C03680=1105.815,151.966,-63.092,-179.395,8.807,149.540
C03681=1105.819,151.717,-63.070,-179.397,8.804,149.540
C03682=1105.824,151.467,-63.048,-179.399,8.800,149.540
C03683=1105.829,151.219,-63.025,-179.401,8.797,149.539
C03684=1105.833,150.970,-63.003,-179.403,8.794,149.539
C03685=1105.838,150.721,-62.980,-179.405,8.790,149.539
C03686=1105.843,150.472,-62.958,-179.407,8.787,149.539
C03687=1105.847,150.223,-62.936,-179.409,8.783,149.538
C03688=1105.852,149.974,-62.913,-179.410,8.781,149.538
C03689=1105.856,149.725,-62.891,-179.413,8.777,149.538
C03690=1105.861,149.476,-62.869,-179.415,8.774,149.538
C03691=1105.865,149.228,-62.847,-179.417,8.770,149.537
C03692=1105.870,148.978,-62.824,-179.418,8.766,149.537
C03693=1105.875,148.729,-62.802,-179.420,8.764,149.537
C03694=1105.879,148.480,-62.780,-179.422,8.760,149.536
C03695=1105.883,148.231,-62.757,-179.424,8.757,149.536
C03696=1105.889,147.982,-62.735,-179.426,8.753,149.536
C03697=1105.893,147.733,-62.713,-179.428,8.749,149.536
C03698=1105.898,147.484,-62.691,-179.430,8.746,149.535
C03699=1105.902,147.236,-62.669,-179.431,8.743,149.535
C03700=1105.908,146.987,-62.646,-179.433,8.740,149.535
C03701=1105.911,146.773,-62.628,-179.435,8.736,149.535
C03702=1105.915,146.560,-62.608,-179.436,8.733,149.534
C03703=1105.919,146.347,-62.590,-179.438,8.730,149.534
C03704=1105.923,146.133,-62.570,-179.439,8.728,149.534
C03705=1105.927,145.920,-62.552,-179.441,8.724,149.533
C03706=1105.931,145.707,-62.533,-179.443,8.721,149.533
C03707=1105.935,145.493,-62.514,-179.444,8.719,149.533
C03708=1105.939,145.280,-62.495,-179.446,8.715,149.533
C03709=1105.943,145.031,-62.473,-179.448,8.711,149.532
C03710=1105.948,144.782,-62.451,-179.449,8.708,149.532
C03711=1105.953,144.533,-62.429,-179.451,8.705,149.532
C03712=1105.957,144.284,-62.408,-179.453,8.701,149.531
C03713=1105.962,144.035,-62.385,-179.455,8.697,149.531
C03714=1105.967,143.787,-62.364,-179.456,8.695,149.531
C03715=1105.972,143.537,-62.341,-179.458,8.691,149.530
C03716=1105.976,143.288,-62.319,-179.460,8.687,149.530
C03717=1105.981,143.039,-62.297,-179.462,8.683,149.530
C03718=1105.986,142.790,-62.276,-179.464,8.680,149.529
C03719=1105.990,142.541,-62.254,-179.465,8.677,149.529
C03720=1105.995,142.292,-62.232,-179.467,8.673,149.529
C03721=1105.999,142.043,-62.210,-179.469,8.670,149.528
C03722=1106.004,141.794,-62.188,-179.470,8.666,149.528
C03723=1106.009,141.546,-62.167,-179.472,8.663,149.528
C03724=1106.013,141.296,-62.145,-179.474,8.660,149.528
C03725=1106.018,141.048,-62.123,-179.476,8.656,149.527
C03726=1106.022,140.798,-62.101,-179.478,8.652,149.527
C03727=1106.027,140.550,-62.079,-179.479,8.650,149.527
C03728=1106.031,140.300,-62.057,-179.481,8.646,149.526
C03729=1106.036,140.052,-62.035,-179.483,8.642,149.526
C03730=1106.040,139.802,-62.013,-179.485,8.639,149.526
C03731=1106.046,139.553,-61.992,-179.486,8.636,149.525
C03732=1106.050,139.304,-61.971,-179.488,8.632,149.525
C03733=1106.055,139.055,-61.949,-179.490,8.629,149.525
C03734=1106.060,138.806,-61.927,-179.491,8.626,149.524
C03735=1106.064,138.557,-61.905,-179.493,8.622,149.524
C03736=1106.069,138.308,-61.883,-179.495,8.619,149.524
C03737=1106.074,138.059,-61.862,-179.497,8.615,149.523
C03738=1106.078,137.810,-61.840,-179.498,8.612,149.523
C03739=1106.082,137.562,-61.819,-179.500,8.609,149.523
C03740=1106.087,137.312,-61.797,-179.502,8.605,149.523
C03741=1106.092,137.063,-61.776,-179.504,8.601,149.522
C03742=1106.097,136.814,-61.754,-179.505,8.599,149.522
C03743=1106.101,136.565,-61.732,-179.507,8.595,149.522
C03744=1106.106,136.316,-61.711,-179.509,8.591,149.521
C03745=1106.111,136.067,-61.690,-179.511,8.589,149.521
C03746=1106.115,135.818,-61.668,-179.512,8.585,149.521
C03747=1106.120,135.569,-61.646,-179.514,8.581,149.521
C03748=1106.125,135.320,-61.626,-179.516,8.578,149.520
C03749=1106.129,135.071,-61.604,-179.518,8.575,149.520
C03750=1106.134,134.822,-61.582,-179.519,8.571,149.520
C03751=1106.139,134.573,-61.561,-179.522,8.568,149.519
C03752=1106.143,134.324,-61.539,-179.523,8.565,149.519
C03753=1106.148,134.075,-61.517,-179.525,8.561,149.519
C03754=1106.152,133.826,-61.497,-179.527,8.558,149.518
C03755=1106.157,133.577,-61.475,-179.529,8.554,149.518
C03756=1106.162,133.327,-61.454,-179.530,8.551,149.518
C03757=1106.166,133.114,-61.436,-179.532,8.549,149.518
C03758=1106.170,132.901,-61.418,-179.533,8.545,149.517
C03759=1106.174,132.688,-61.399,-179.535,8.542,149.517
C03760=1106.178,132.474,-61.381,-179.536,8.539,149.517
C03761=1106.182,132.261,-61.362,-179.538,8.537,149.517
C03762=1106.186,132.047,-61.344,-179.539,8.534,149.516
C03763=1106.190,131.834,-61.326,-179.540,8.531,149.516
C03764=1106.194,131.621,-61.308,-179.543,8.528,149.516
C03765=1106.199,131.372,-61.287,-179.544,8.525,149.516
C03766=1106.203,131.122,-61.265,-179.546,8.521,149.516
C03767=1106.208,130.873,-61.244,-179.548,8.518,149.515
C03768=1106.212,130.625,-61.223,-179.549,8.515,149.515
C03769=1106.217,130.376,-61.202,-179.551,8.511,149.515
C03770=1106.222,130.126,-61.180,-179.553,8.508,149.514
C03771=1106.226,129.877,-61.159,-179.554,8.505,149.514
C03772=1106.231,129.629,-61.138,-179.556,8.501,149.514
C03773=1106.236,129.379,-61.117,-179.558,8.498,149.513
C03774=1106.241,129.130,-61.096,-179.560,8.495,149.513
C03775=1106.245,128.881,-61.074,-179.561,8.491,149.513
C03776=1106.250,128.632,-61.053,-179.564,8.488,149.513
C03777=1106.255,128.383,-61.033,-179.566,8.484,149.512
C03778=1106.259,128.134,-61.011,-179.567,8.481,149.512
C03779=1106.265,127.885,-60.990,-179.569,8.478,149.512
C03780=1106.268,127.635,-60.970,-179.571,8.474,149.511
C03781=1106.273,127.387,-60.948,-179.572,8.471,149.511
C03782=1106.278,127.137,-60.927,-179.574,8.468,149.511
C03783=1106.283,126.889,-60.907,-179.576,8.464,149.511
C03784=1106.288,126.640,-60.885,-179.577,8.461,149.510
C03785=1106.292,126.391,-60.865,-179.579,8.458,149.510
C03786=1106.297,126.141,-60.843,-179.581,8.454,149.510
C03787=1106.302,125.892,-60.822,-179.582,8.451,149.509
C03788=1106.306,125.643,-60.801,-179.585,8.448,149.509
C03789=1106.311,125.394,-60.780,-179.587,8.444,149.509
C03790=1106.316,125.145,-60.760,-179.588,8.442,149.509
C03791=1106.321,124.896,-60.739,-179.590,8.438,149.508
C03792=1106.325,124.648,-60.718,-179.592,8.434,149.508
C03793=1106.330,124.398,-60.696,-179.593,8.431,149.508
C03794=1106.334,124.149,-60.676,-179.595,8.428,149.508
C03795=1106.339,123.899,-60.655,-179.597,8.424,149.507
C03796=1106.344,123.650,-60.635,-179.598,8.421,149.507
C03797=1106.349,123.401,-60.614,-179.600,8.418,149.507
C03798=1106.353,123.153,-60.593,-179.602,8.414,149.506
C03799=1106.358,122.904,-60.572,-179.603,8.411,149.506
C03800=1106.363,122.655,-60.551,-179.605,8.408,149.506
C03801=1106.368,122.405,-60.530,-179.608,8.404,149.506
C03802=1106.372,122.156,-60.510,-179.609,8.402,149.505
C03803=1106.376,121.907,-60.489,-179.611,8.398,149.505
C03804=1106.381,121.658,-60.468,-179.613,8.394,149.505
C03805=1106.386,121.409,-60.448,-179.614,8.391,149.504
C03806=1106.391,121.159,-60.427,-179.616,8.388,149.504
C03807=1106.395,120.910,-60.407,-179.618,8.384,149.504
C03808=1106.400,120.661,-60.386,-179.620,8.381,149.504
C03809=1106.405,120.412,-60.365,-179.621,8.378,149.503
C03810=1106.409,120.163,-60.345,-179.623,8.374,149.503
C03811=1106.414,119.914,-60.324,-179.625,8.370,149.503
C03812=1106.419,119.665,-60.304,-179.626,8.368,149.502
C03813=1106.423,119.452,-60.285,-179.628,8.365,149.502
C03814=1106.427,119.238,-60.268,-179.630,8.362,149.502
C03815=1106.431,119.025,-60.250,-179.631,8.359,149.502
C03816=1106.435,118.811,-60.232,-179.633,8.356,149.502
C03817=1106.439,118.598,-60.216,-179.634,8.353,149.501
C03818=1106.443,118.385,-60.198,-179.635,8.350,149.501
C03819=1106.447,118.171,-60.180,-179.637,8.348,149.501
C03820=1106.451,117.958,-60.162,-179.638,8.345,149.500
C03821=1106.456,117.708,-60.142,-179.640,8.341,149.500
C03822=1106.461,117.459,-60.121,-179.642,8.338,149.500
C03823=1106.465,117.210,-60.101,-179.644,8.334,149.500
C03824=1106.470,116.961,-60.081,-179.645,8.331,149.499
C03825=1106.475,116.712,-60.060,-179.647,8.328,149.499
C03826=1106.479,116.463,-60.039,-179.649,8.324,149.499
C03827=1106.484,116.214,-60.019,-179.650,8.321,149.498
C03828=1106.488,115.964,-59.999,-179.652,8.318,149.498
C03829=1106.494,115.715,-59.978,-179.654,8.314,149.498
C03830=1106.498,115.466,-59.958,-179.655,8.311,149.498
C03831=1106.503,115.218,-59.938,-179.658,8.308,149.497
C03832=1106.508,114.969,-59.918,-179.659,8.304,149.497
C03833=1106.513,114.719,-59.897,-179.661,8.301,149.497
C03834=1106.518,114.470,-59.877,-179.663,8.297,149.496
C03835=1106.522,114.221,-59.857,-179.664,8.294,149.496
C03836=1106.526,113.972,-59.836,-179.666,8.291,149.496
C03837=1106.532,113.722,-59.816,-179.668,8.287,149.496
C03838=1106.536,113.473,-59.796,-179.669,8.283,149.495
C03839=1106.541,113.224,-59.775,-179.671,8.280,149.495
C03840=1106.545,112.975,-59.756,-179.672,8.277,149.494
C03841=1106.550,112.726,-59.735,-179.674,8.273,149.494
C03842=1106.555,112.476,-59.714,-179.677,8.270,149.494
C03843=1106.560,112.228,-59.695,-179.678,8.267,149.494
C03844=1106.565,111.979,-59.675,-179.680,8.263,149.493
C03845=1106.569,111.730,-59.654,-179.681,8.259,149.493
C03846=1106.574,111.480,-59.634,-179.683,8.257,149.493
C03847=1106.578,111.231,-59.614,-179.685,8.253,149.492
C03848=1106.583,110.982,-59.594,-179.686,8.249,149.492
C03849=1106.588,110.732,-59.573,-179.688,8.246,149.492
C03850=1106.593,110.484,-59.553,-179.690,8.242,149.492
C03851=1106.598,110.235,-59.534,-179.692,8.238,149.491
C03852=1106.603,109.986,-59.513,-179.694,8.235,149.491
C03853=1106.607,109.736,-59.494,-179.696,8.231,149.491
C03854=1106.612,109.487,-59.473,-179.698,8.228,149.490
C03855=1106.617,109.237,-59.454,-179.699,8.225,149.490
C03856=1106.622,108.989,-59.434,-179.701,8.221,149.490
C03857=1106.626,108.740,-59.414,-179.703,8.217,149.489
C03858=1106.631,108.491,-59.394,-179.705,8.214,149.489
C03859=1106.636,108.241,-59.374,-179.706,8.210,149.489
C03860=1106.640,107.992,-59.354,-179.709,8.207,149.488
C03861=1106.645,107.743,-59.334,-179.710,8.203,149.488
C03862=1106.650,107.494,-59.315,-179.712,8.199,149.488
C03863=1106.654,107.245,-59.294,-179.714,8.195,149.487
C03864=1106.659,106.995,-59.275,-179.716,8.192,149.487
C03865=1106.664,106.746,-59.254,-179.717,8.188,149.487
C03866=1106.669,106.497,-59.235,-179.719,8.185,149.486
C03867=1106.674,106.248,-59.215,-179.721,8.181,149.486
C03868=1106.678,105.999,-59.195,-179.723,8.178,149.486
C03869=1106.682,105.785,-59.178,-179.724,8.174,149.485
C03870=1106.686,105.572,-59.161,-179.726,8.171,149.485
C03871=1106.691,105.358,-59.144,-179.727,8.168,149.485
C03872=1106.695,105.144,-59.127,-179.729,8.165,149.484
C03873=1106.699,104.931,-59.110,-179.730,8.162,149.484
C03874=1106.703,104.717,-59.093,-179.731,8.159,149.484
C03875=1106.707,104.504,-59.076,-179.733,8.155,149.484
C03876=1106.711,104.290,-59.059,-179.734,8.152,149.483
C03877=1106.715,104.041,-59.040,-179.736,8.149,149.483
C03878=1106.720,103.792,-59.020,-179.738,8.145,149.482
C03879=1106.726,103.543,-59.001,-179.739,8.142,149.482
C03880=1106.730,103.294,-58.981,-179.741,8.138,149.482
C03881=1106.735,103.044,-58.961,-179.742,8.134,149.481
C03882=1106.740,102.795,-58.942,-179.744,8.130,149.481
C03883=1106.745,102.546,-58.922,-179.746,8.126,149.480
C03884=1106.749,102.297,-58.902,-179.747,8.123,149.480
C03885=1106.753,102.048,-58.883,-179.749,8.119,149.480
C03886=1106.759,101.799,-58.863,-179.751,8.115,149.479
C03887=1106.763,101.549,-58.844,-179.752,8.112,149.479
C03888=1106.768,101.299,-58.824,-179.753,8.108,149.479
C03889=1106.773,101.051,-58.805,-179.755,8.104,149.478
C03890=1106.778,100.802,-58.784,-179.757,8.100,149.478
C03891=1106.782,100.552,-58.765,-179.759,8.097,149.477
C03892=1106.787,100.304,-58.746,-179.760,8.093,149.477
C03893=1106.792,100.054,-58.726,-179.761,8.090,149.477
C03894=1106.797,99.805,-58.707,-179.763,8.086,149.476
C03895=1106.802,99.556,-58.687,-179.764,8.082,149.476
C03896=1106.806,99.306,-58.668,-179.766,8.078,149.475
C03897=1106.811,99.057,-58.649,-179.768,8.074,149.475
C03898=1106.816,98.808,-58.629,-179.769,8.070,149.474
C03899=1106.821,98.558,-58.610,-179.770,8.067,149.474
C03900=1106.825,98.310,-58.591,-179.772,8.063,149.473
C03901=1106.830,98.060,-58.571,-179.773,8.060,149.473
C03902=1106.836,97.811,-58.552,-179.775,8.056,149.473
C03903=1106.840,97.562,-58.533,-179.777,8.052,149.472
C03904=1106.844,97.312,-58.513,-179.778,8.049,149.472
C03905=1106.850,97.064,-58.494,-179.779,8.045,149.471
C03906=1106.854,96.814,-58.474,-179.781,8.041,149.471
C03907=1106.859,96.565,-58.456,-179.782,8.037,149.470
C03908=1106.864,96.316,-58.436,-179.784,8.033,149.470
C03909=1106.869,96.066,-58.416,-179.785,8.030,149.470
C03910=1106.873,95.818,-58.398,-179.787,8.026,149.469
C03911=1106.878,95.568,-58.378,-179.788,8.022,149.469
C03912=1106.883,95.319,-58.359,-179.790,8.018,149.468
C03913=1106.887,95.070,-58.340,-179.791,8.014,149.468
C03914=1106.893,94.821,-58.321,-179.792,8.011,149.467
C03915=1106.897,94.571,-58.302,-179.794,8.007,149.467
C03916=1106.902,94.322,-58.283,-179.795,8.003,149.466
C03917=1106.907,94.073,-58.263,-179.797,7.999,149.466
C03918=1106.912,93.824,-58.244,-179.798,7.996,149.465
C03919=1106.916,93.575,-58.225,-179.799,7.992,149.465
C03920=1106.921,93.325,-58.206,-179.800,7.988,149.464
C03921=1106.926,93.076,-58.187,-179.802,7.984,149.464
C03922=1106.931,92.826,-58.167,-179.803,7.981,149.463
C03923=1106.935,92.578,-58.149,-179.805,7.977,149.463
C03924=1106.940,92.328,-58.129,-179.806,7.973,149.462
C03925=1106.944,92.115,-58.113,-179.807,7.970,149.462
C03926=1106.948,91.901,-58.097,-179.808,7.967,149.462
C03927=1106.952,91.688,-58.081,-179.809,7.964,149.461
C03928=1106.957,91.474,-58.064,-179.811,7.960,149.461
C03929=1106.961,91.260,-58.048,-179.812,7.957,149.460
C03930=1106.965,91.047,-58.032,-179.813,7.954,149.460
C03931=1106.969,90.833,-58.015,-179.814,7.951,149.460
C03932=1106.973,90.619,-58.000,-179.815,7.948,149.459
C03933=1106.978,90.370,-57.980,-179.816,7.944,149.459
C03934=1106.983,90.121,-57.962,-179.817,7.940,149.458
C03935=1106.988,89.871,-57.942,-179.819,7.936,149.458
C03936=1106.992,89.622,-57.924,-179.820,7.933,149.457
C03937=1106.998,89.373,-57.905,-179.821,7.928,149.457
C03938=1107.002,89.124,-57.886,-179.823,7.924,149.456
C03939=1107.007,88.875,-57.867,-179.824,7.921,149.456
C03940=1107.011,88.625,-57.848,-179.825,7.917,149.455
C03941=1107.017,88.376,-57.829,-179.826,7.913,149.455
C03942=1107.021,88.127,-57.810,-179.827,7.910,149.454
C03943=1107.026,87.877,-57.792,-179.828,7.906,149.453
C03944=1107.031,87.629,-57.773,-179.830,7.902,149.453
C03945=1107.035,87.379,-57.755,-179.831,7.899,149.453
C03946=1107.041,87.130,-57.735,-179.832,7.894,149.452
C03947=1107.045,86.880,-57.717,-179.834,7.891,149.452
C03948=1107.050,86.631,-57.698,-179.834,7.887,149.451
C03949=1107.055,86.382,-57.680,-179.836,7.883,149.450
C03950=1107.059,86.133,-57.661,-179.837,7.879,149.450
C03951=1107.065,85.883,-57.642,-179.838,7.876,149.449
C03952=1107.069,85.634,-57.623,-179.840,7.872,149.449
C03953=1107.075,85.385,-57.604,-179.840,7.868,149.448
C03954=1107.079,85.136,-57.586,-179.842,7.864,149.448
C03955=1107.083,84.886,-57.567,-179.843,7.860,149.447
C03956=1107.089,84.637,-57.548,-179.844,7.857,149.447
C03957=1107.094,84.388,-57.530,-179.845,7.853,149.446
C03958=1107.098,84.139,-57.511,-179.846,7.850,149.446
C03959=1107.103,83.889,-57.492,-179.847,7.846,149.445
C03960=1107.107,83.640,-57.473,-179.849,7.842,149.445
C03961=1107.112,83.391,-57.455,-179.849,7.838,149.444
C03962=1107.118,83.142,-57.437,-179.851,7.834,149.444
C03963=1107.122,82.892,-57.418,-179.852,7.831,149.443
C03964=1107.127,82.643,-57.400,-179.853,7.827,149.442
C03965=1107.132,82.394,-57.382,-179.854,7.824,149.442
C03966=1107.137,82.144,-57.362,-179.855,7.819,149.441
C03967=1107.141,81.895,-57.344,-179.856,7.815,149.441
C03968=1107.146,81.647,-57.325,-179.857,7.812,149.440
C03969=1107.152,81.397,-57.307,-179.858,7.808,149.440
C03970=1107.156,81.147,-57.288,-179.859,7.805,149.439
C03971=1107.161,80.898,-57.271,-179.861,7.801,149.439
C03972=1107.166,80.650,-57.252,-179.861,7.797,149.438
C03973=1107.171,80.399,-57.233,-179.863,7.793,149.438
C03974=1107.176,80.150,-57.215,-179.863,7.790,149.437
C03975=1107.180,79.902,-57.196,-179.864,7.786,149.436
C03976=1107.185,79.652,-57.178,-179.865,7.782,149.436
C03977=1107.189,79.403,-57.160,-179.866,7.778,149.435
C03978=1107.195,79.153,-57.141,-179.867,7.775,149.435
C03979=1107.200,78.905,-57.123,-179.868,7.771,149.434
C03980=1107.204,78.655,-57.104,-179.869,7.768,149.434
C03981=1107.208,78.441,-57.089,-179.870,7.764,149.433
C03982=1107.213,78.228,-57.073,-179.871,7.761,149.433
C03983=1107.217,78.013,-57.057,-179.872,7.758,149.432
C03984=1107.221,77.800,-57.042,-179.873,7.755,149.432
C03985=1107.225,77.586,-57.026,-179.874,7.752,149.431
C03986=1107.229,77.373,-57.010,-179.874,7.748,149.431
C03987=1107.233,77.159,-56.995,-179.875,7.745,149.430
C03988=1107.237,76.944,-56.979,-179.876,7.742,149.430
C03989=1107.242,76.696,-56.961,-179.878,7.738,149.429
C03990=1107.247,76.447,-56.943,-179.879,7.734,149.429
C03991=1107.252,76.197,-56.924,-179.880,7.730,149.428
C03992=1107.257,75.947,-56.906,-179.882,7.726,149.428
C03993=1107.262,75.698,-56.888,-179.884,7.722,149.427
C03994=1107.267,75.449,-56.870,-179.885,7.718,149.427
C03995=1107.272,75.200,-56.852,-179.886,7.715,149.426
C03996=1107.276,74.951,-56.834,-179.887,7.711,149.426
C03997=1107.281,74.701,-56.815,-179.888,7.706,149.425
C03998=1107.285,74.452,-56.797,-179.890,7.703,149.425
C03999=1107.290,74.203,-56.779,-179.892,7.699,149.424
C04000=1107.295,73.954,-56.761,-179.893,7.695,149.424
C04001=1107.300,73.705,-56.743,-179.894,7.690,149.423
C04002=1107.305,73.455,-56.724,-179.896,7.687,149.423
C04003=1107.310,73.205,-56.706,-179.897,7.683,149.422
C04004=1107.315,72.956,-56.688,-179.899,7.678,149.422
C04005=1107.320,72.707,-56.670,-179.899,7.675,149.421
C04006=1107.325,72.458,-56.652,-179.901,7.671,149.421
C04007=1107.330,72.209,-56.634,-179.902,7.667,149.420
C04008=1107.335,71.959,-56.617,-179.904,7.663,149.420
C04009=1107.339,71.709,-56.598,-179.905,7.659,149.419
C04010=1107.344,71.460,-56.580,-179.906,7.655,149.419
C04011=1107.349,71.211,-56.562,-179.908,7.651,149.418
C04012=1107.354,70.961,-56.544,-179.910,7.647,149.418
C04013=1107.359,70.712,-56.526,-179.911,7.643,149.417
C04014=1107.364,70.463,-56.508,-179.912,7.640,149.417
C04015=1107.368,70.214,-56.491,-179.913,7.636,149.416
C04016=1107.373,69.965,-56.473,-179.914,7.632,149.416
C04017=1107.378,69.716,-56.455,-179.916,7.628,149.415
C04018=1107.382,69.465,-56.438,-179.917,7.624,149.415
C04019=1107.387,69.216,-56.420,-179.919,7.620,149.414
C04020=1107.392,68.967,-56.402,-179.920,7.616,149.414
C04021=1107.397,68.718,-56.384,-179.921,7.613,149.413
C04022=1107.402,68.469,-56.366,-179.922,7.608,149.413
C04023=1107.407,68.219,-56.348,-179.924,7.604,149.412
C04024=1107.412,67.970,-56.330,-179.925,7.600,149.412
C04025=1107.417,67.721,-56.312,-179.926,7.596,149.411
C04026=1107.421,67.472,-56.295,-179.928,7.592,149.411
C04027=1107.427,67.222,-56.278,-179.930,7.588,149.410
C04028=1107.431,66.973,-56.260,-179.930,7.585,149.410
C04029=1107.436,66.724,-56.242,-179.932,7.581,149.409
C04030=1107.441,66.474,-56.224,-179.933,7.577,149.409
C04031=1107.446,66.225,-56.207,-179.934,7.573,149.408
C04032=1107.451,65.976,-56.189,-179.936,7.569,149.408
C04033=1107.456,65.727,-56.171,-179.937,7.565,149.407
C04034=1107.461,65.477,-56.154,-179.939,7.561,149.407
C04035=1107.466,65.228,-56.136,-179.939,7.557,149.406
C04036=1107.471,64.978,-56.118,-179.941,7.553,149.406
C04037=1107.474,64.764,-56.103,-179.942,7.549,149.405
C04038=1107.479,64.550,-56.088,-179.943,7.546,149.405
C04039=1107.482,64.337,-56.073,-179.944,7.543,149.404
C04040=1107.487,64.123,-56.058,-179.945,7.540,149.404
C04041=1107.492,63.909,-56.043,-179.947,7.536,149.403
C04042=1107.495,63.695,-56.027,-179.948,7.533,149.403
C04043=1107.500,63.481,-56.012,-179.948,7.529,149.402
C04044=1107.504,63.267,-55.998,-179.950,7.526,149.402
C04045=1107.509,63.018,-55.980,-179.951,7.522,149.401
C04046=1107.514,62.768,-55.963,-179.952,7.518,149.401
C04047=1107.518,62.520,-55.945,-179.953,7.514,149.400
C04048=1107.523,62.270,-55.928,-179.955,7.510,149.400
C04049=1107.528,62.021,-55.910,-179.956,7.506,149.399
C04050=1107.533,61.771,-55.893,-179.957,7.502,149.399
C04051=1107.537,61.522,-55.875,-179.958,7.499,149.398
C04052=1107.543,61.272,-55.858,-179.959,7.495,149.398
C04053=1107.548,61.023,-55.840,-179.961,7.490,149.397
C04054=1107.552,60.773,-55.824,-179.962,7.486,149.397
C04055=1107.558,60.525,-55.806,-179.963,7.482,149.396
C04056=1107.563,60.275,-55.789,-179.964,7.479,149.396
C04057=1107.567,60.026,-55.771,-179.965,7.475,149.395
C04058=1107.572,59.776,-55.754,-179.967,7.471,149.394
C04059=1107.576,59.528,-55.737,-179.968,7.467,149.394
C04060=1107.582,59.278,-55.719,-179.969,7.463,149.393
C04061=1107.587,59.028,-55.702,-179.970,7.459,149.393
C04062=1107.591,58.779,-55.685,-179.972,7.455,149.392
C04063=1107.596,58.529,-55.667,-179.973,7.451,149.392
C04064=1107.601,58.280,-55.649,-179.974,7.447,149.391
C04065=1107.606,58.031,-55.633,-179.975,7.443,149.391
C04066=1107.611,57.782,-55.616,-179.977,7.439,149.390
C04067=1107.616,57.533,-55.599,-179.977,7.435,149.389
C04068=1107.621,57.283,-55.581,-179.979,7.431,149.389
C04069=1107.626,57.033,-55.564,-179.980,7.427,149.388
C04070=1107.630,56.784,-55.547,-179.982,7.423,149.388
C04071=1107.636,56.535,-55.530,-179.983,7.419,149.387
C04072=1107.640,56.286,-55.513,-179.984,7.416,149.387
C04073=1107.646,56.036,-55.496,-179.985,7.412,149.386
C04074=1107.650,55.787,-55.478,-179.986,7.407,149.386
C04075=1107.655,55.537,-55.461,-179.987,7.403,149.385
C04076=1107.660,55.288,-55.444,-179.988,7.400,149.384
C04077=1107.665,55.039,-55.428,-179.989,7.396,149.384
C04078=1107.670,54.790,-55.410,-179.990,7.392,149.383
C04079=1107.675,54.540,-55.393,-179.992,7.388,149.383
C04080=1107.679,54.291,-55.376,-179.993,7.383,149.382
C04081=1107.684,54.041,-55.359,-179.994,7.380,149.382
C04082=1107.690,53.792,-55.343,-179.995,7.376,149.381
C04083=1107.694,53.543,-55.325,-179.996,7.372,149.381
C04084=1107.699,53.293,-55.308,-179.998,7.368,149.380
C04085=1107.704,53.044,-55.291,-179.999,7.363,149.379
C04086=1107.709,52.795,-55.274,-179.999,7.360,149.379
C04087=1107.714,52.545,-55.257,179.999,7.356,149.378
C04088=1107.719,52.295,-55.241,179.998,7.352,149.378
C04089=1107.724,52.046,-55.223,179.997,7.347,149.377
C04090=1107.728,51.797,-55.206,179.996,7.344,149.377
C04091=1107.734,51.548,-55.189,179.995,7.340,149.376
C04092=1107.739,51.298,-55.172,179.994,7.336,149.375
C04093=1107.743,51.085,-55.158,179.993,7.333,149.375
C04094=1107.747,50.870,-55.144,179.991,7.329,149.374
C04095=1107.752,50.656,-55.129,179.990,7.326,149.374
C04096=1107.756,50.442,-55.115,179.990,7.322,149.373
C04097=1107.760,50.229,-55.100,179.989,7.319,149.373
C04098=1107.764,50.015,-55.086,179.988,7.316,149.372
C04099=1107.769,49.800,-55.072,179.987,7.312,149.372
C04100=1107.773,49.587,-55.057,179.986,7.308,149.371
C04101=1107.777,49.337,-55.041,179.985,7.304,149.371
C04102=1107.782,49.087,-55.023,179.984,7.301,149.370
C04103=1107.787,48.839,-55.007,179.983,7.297,149.370
C04104=1107.792,48.589,-54.990,179.982,7.292,149.369
C04105=1107.797,48.339,-54.973,179.980,7.288,149.369
C04106=1107.802,48.091,-54.957,179.979,7.284,149.368
C04107=1107.807,47.841,-54.940,179.979,7.281,149.367
C04108=1107.811,47.592,-54.923,179.978,7.276,149.367
C04109=1107.816,47.342,-54.906,179.976,7.272,149.366
C04110=1107.821,47.093,-54.890,179.975,7.268,149.365
C04111=1107.826,46.844,-54.873,179.975,7.265,149.365
C04112=1107.831,46.594,-54.856,179.974,7.260,149.364
C04113=1107.837,46.344,-54.840,179.972,7.256,149.364
C04114=1107.841,46.095,-54.824,179.971,7.252,149.363
C04115=1107.845,45.845,-54.807,179.970,7.249,149.362
C04116=1107.851,45.596,-54.790,179.969,7.244,149.362
C04117=1107.856,45.347,-54.773,179.968,7.240,149.361
C04118=1107.861,45.098,-54.757,179.967,7.236,149.361
C04119=1107.865,44.849,-54.740,179.966,7.233,149.360
C04120=1107.871,44.598,-54.724,179.965,7.228,149.359
C04121=1107.876,44.349,-54.708,179.964,7.224,149.359
C04122=1107.880,44.100,-54.691,179.963,7.220,149.358
C04123=1107.885,43.850,-54.674,179.962,7.217,149.358
C04124=1107.890,43.602,-54.658,179.961,7.212,149.357
C04125=1107.896,43.351,-54.641,179.960,7.208,149.356
C04126=1107.901,43.102,-54.625,179.959,7.204,149.356
C04127=1107.905,42.853,-54.608,179.958,7.200,149.355
C04128=1107.910,42.603,-54.592,179.957,7.196,149.355
C04129=1107.915,42.354,-54.576,179.956,7.192,149.354
C04130=1107.919,42.105,-54.559,179.955,7.188,149.353
C04131=1107.925,41.855,-54.543,179.954,7.184,149.353
C04132=1107.930,41.605,-54.527,179.953,7.180,149.352
C04133=1107.935,41.357,-54.510,179.952,7.175,149.351
C04134=1107.940,41.107,-54.494,179.951,7.171,149.351
C04135=1107.945,40.858,-54.478,179.951,7.168,149.350
C04136=1107.949,40.608,-54.461,179.949,7.164,149.350
C04137=1107.954,40.359,-54.445,179.948,7.159,149.349
C04138=1107.960,40.109,-54.429,179.947,7.155,149.348
C04139=1107.965,39.860,-54.412,179.946,7.152,149.348
C04140=1107.970,39.611,-54.396,179.945,7.147,149.347
C04141=1107.974,39.361,-54.380,179.944,7.143,149.346
C04142=1107.979,39.112,-54.363,179.943,7.139,149.346
C04143=1107.984,38.862,-54.347,179.943,7.135,149.345
C04144=1107.989,38.613,-54.331,179.942,7.131,149.344
C04145=1107.994,38.364,-54.314,179.941,7.127,149.344
C04146=1107.999,38.114,-54.299,179.940,7.122,149.343
C04147=1108.004,37.865,-54.282,179.939,7.119,149.342
C04148=1108.009,37.615,-54.267,179.938,7.114,149.342
C04149=1108.013,37.402,-54.252,179.937,7.111,149.341
C04150=1108.017,37.187,-54.238,179.936,7.107,149.341
C04151=1108.022,36.973,-54.225,179.936,7.104,149.340
C04152=1108.026,36.759,-54.210,179.935,7.100,149.340
C04153=1108.030,36.545,-54.197,179.934,7.097,149.339
C04154=1108.035,36.331,-54.183,179.933,7.094,149.338
C04155=1108.039,36.117,-54.170,179.932,7.089,149.338
C04156=1108.043,35.903,-54.155,179.931,7.086,149.337
C04157=1108.048,35.653,-54.139,179.930,7.082,149.337
C04158=1108.053,35.404,-54.123,179.930,7.078,149.336
C04159=1108.058,35.155,-54.107,179.929,7.074,149.335
C04160=1108.063,34.905,-54.091,179.928,7.069,149.335
C04161=1108.068,34.656,-54.075,179.927,7.065,149.334
C04162=1108.073,34.406,-54.059,179.927,7.062,149.333
C04163=1108.078,34.157,-54.043,179.926,7.057,149.333
C04164=1108.083,33.907,-54.027,179.925,7.053,149.332
C04165=1108.088,33.658,-54.010,179.924,7.049,149.331
C04166=1108.093,33.409,-53.995,179.923,7.045,149.331
C04167=1108.097,33.159,-53.980,179.922,7.041,149.330
C04168=1108.102,32.910,-53.963,179.921,7.037,149.329
C04169=1108.107,32.660,-53.947,179.920,7.032,149.329
C04170=1108.113,32.411,-53.932,179.920,7.028,149.328
C04171=1108.118,32.162,-53.915,179.919,7.024,149.327
C04172=1108.123,31.912,-53.899,179.918,7.020,149.326
C04173=1108.128,31.662,-53.884,179.917,7.015,149.326
C04174=1108.132,31.413,-53.867,179.916,7.012,149.325
C04175=1108.137,31.164,-53.852,179.915,7.008,149.324
C04176=1108.142,30.915,-53.837,179.914,7.003,149.324
C04177=1108.147,30.664,-53.821,179.914,6.999,149.323
C04178=1108.152,30.416,-53.804,179.913,6.995,149.322
C04179=1108.157,30.166,-53.788,179.912,6.991,149.322
C04180=1108.162,29.916,-53.773,179.911,6.986,149.321
C04181=1108.168,29.667,-53.757,179.911,6.983,149.320
C04182=1108.172,29.418,-53.741,179.910,6.978,149.319
C04183=1108.177,29.168,-53.726,179.909,6.974,149.319
C04184=1108.182,28.919,-53.710,179.908,6.970,149.318
C04185=1108.187,28.669,-53.694,179.907,6.966,149.317
C04186=1108.192,28.420,-53.678,179.907,6.961,149.317
C04187=1108.197,28.171,-53.663,179.906,6.957,149.316
C04188=1108.202,27.921,-53.647,179.905,6.953,149.315
C04189=1108.207,27.671,-53.631,179.904,6.949,149.315
C04190=1108.212,27.422,-53.616,179.904,6.945,149.314
C04191=1108.217,27.172,-53.600,179.903,6.940,149.313
C04192=1108.222,26.923,-53.585,179.902,6.936,149.312
C04193=1108.227,26.674,-53.568,179.902,6.932,149.312
C04194=1108.232,26.424,-53.552,179.901,6.928,149.311
C04195=1108.236,26.175,-53.537,179.900,6.923,149.310
C04196=1108.242,25.925,-53.522,179.899,6.919,149.309
C04197=1108.247,25.676,-53.506,179.899,6.915,149.309
C04198=1108.252,25.426,-53.490,179.897,6.911,149.308
C04199=1108.257,25.177,-53.475,179.897,6.906,149.307
C04200=1108.262,24.927,-53.460,179.896,6.902,149.306
C04201=1108.267,24.677,-53.444,179.895,6.898,149.306
C04202=1108.271,24.428,-53.429,179.895,6.894,149.305
C04203=1108.277,24.179,-53.413,179.894,6.889,149.304
C04204=1108.282,23.929,-53.398,179.893,6.885,149.304
C04205=1108.286,23.715,-53.384,179.892,6.882,149.303
C04206=1108.290,23.501,-53.371,179.892,6.878,149.302
C04207=1108.295,23.287,-53.357,179.891,6.874,149.302
C04208=1108.299,23.073,-53.344,179.891,6.871,149.301
C04209=1108.303,22.859,-53.331,179.890,6.867,149.300
C04210=1108.308,22.645,-53.318,179.890,6.863,149.300
C04211=1108.312,22.431,-53.305,179.889,6.860,149.299
C04212=1108.316,22.216,-53.291,179.889,6.856,149.298
C04213=1108.321,21.967,-53.276,179.888,6.852,149.298
C04214=1108.326,21.718,-53.261,179.887,6.847,149.297
C04215=1108.331,21.469,-53.245,179.886,6.843,149.296
C04216=1108.335,21.219,-53.230,179.886,6.839,149.295
C04217=1108.341,20.969,-53.214,179.885,6.835,149.295
C04218=1108.346,20.719,-53.199,179.884,6.830,149.294
C04219=1108.351,20.470,-53.184,179.883,6.826,149.293
C04220=1108.356,20.220,-53.168,179.883,6.822,149.292
C04221=1108.360,19.971,-53.153,179.882,6.817,149.292
C04222=1108.366,19.722,-53.138,179.882,6.813,149.291
C04223=1108.371,19.473,-53.123,179.881,6.808,149.290
C04224=1108.376,19.223,-53.107,179.881,6.804,149.289
C04225=1108.381,18.974,-53.092,179.880,6.800,149.288
C04226=1108.386,18.723,-53.077,179.879,6.795,149.288
C04227=1108.391,18.474,-53.061,179.879,6.791,149.287
C04228=1108.396,18.225,-53.046,179.878,6.787,149.286
C04229=1108.401,17.975,-53.031,179.878,6.782,149.285
C04230=1108.406,17.726,-53.016,179.877,6.778,149.284
C04231=1108.411,17.476,-53.001,179.876,6.773,149.284
C04232=1108.415,17.226,-52.985,179.876,6.769,149.283
C04233=1108.421,16.977,-52.970,179.875,6.765,149.282
C04234=1108.426,16.728,-52.955,179.875,6.760,149.281
C04235=1108.431,16.478,-52.940,179.874,6.756,149.280
C04236=1108.436,16.229,-52.925,179.874,6.752,149.280
C04237=1108.441,15.979,-52.909,179.873,6.748,149.279
C04238=1108.446,15.730,-52.894,179.872,6.743,149.278
C04239=1108.451,15.481,-52.880,179.871,6.739,149.277
C04240=1108.456,15.231,-52.864,179.871,6.735,149.276
C04241=1108.460,14.981,-52.849,179.871,6.730,149.275
C04242=1108.466,14.731,-52.834,179.870,6.726,149.275
C04243=1108.471,14.482,-52.819,179.869,6.721,149.274
C04244=1108.476,14.233,-52.804,179.869,6.716,149.273
C04245=1108.481,13.983,-52.789,179.869,6.712,149.272
C04246=1108.486,13.734,-52.774,179.868,6.708,149.271
C04247=1108.491,13.485,-52.759,179.867,6.703,149.271
C04248=1108.496,13.235,-52.745,179.867,6.699,149.270
C04249=1108.501,12.986,-52.729,179.867,6.695,149.269
C04250=1108.506,12.736,-52.715,179.866,6.690,149.268
C04251=1108.511,12.487,-52.700,179.865,6.686,149.267
C04252=1108.516,12.237,-52.684,179.865,6.681,149.266
C04253=1108.521,11.987,-52.669,179.864,6.676,149.265
C04254=1108.526,11.738,-52.654,179.864,6.672,149.265
C04255=1108.531,11.488,-52.640,179.863,6.668,149.264
C04256=1108.536,11.239,-52.625,179.862,6.663,149.263
C04257=1108.541,10.989,-52.610,179.862,6.659,149.262
C04258=1108.546,10.740,-52.595,179.862,6.655,149.261
C04259=1108.551,10.491,-52.580,179.861,6.650,149.260
C04260=1108.556,10.241,-52.565,179.861,6.645,149.260
C04261=1108.561,10.027,-52.553,179.860,6.642,149.259
C04262=1108.564,9.813,-52.540,179.861,6.638,149.258
C04263=1108.570,9.598,-52.527,179.860,6.633,149.257
C04264=1108.573,9.384,-52.514,179.859,6.630,149.257
C04265=1108.578,9.170,-52.502,179.859,6.626,149.256
C04266=1108.582,8.956,-52.489,179.859,6.622,149.255
C04267=1108.586,8.742,-52.476,179.858,6.618,149.254
C04268=1108.591,8.527,-52.463,179.858,6.614,149.254
C04269=1108.596,8.278,-52.449,179.857,6.610,149.253
C04270=1108.601,8.028,-52.434,179.857,6.605,149.252
C04271=1108.606,7.779,-52.420,179.856,6.600,149.251
C04272=1108.611,7.529,-52.404,179.855,6.596,149.250
C04273=1108.616,7.280,-52.390,179.855,6.591,149.249
C04274=1108.621,7.031,-52.375,179.854,6.586,149.248
C04275=1108.625,6.781,-52.361,179.854,6.582,149.248
C04276=1108.631,6.531,-52.346,179.852,6.577,149.247
C04277=1108.636,6.282,-52.331,179.852,6.573,149.246
C04278=1108.641,6.032,-52.316,179.851,6.568,149.245
C04279=1108.646,5.782,-52.302,179.851,6.563,149.244
C04280=1108.650,5.533,-52.287,179.850,6.559,149.244
C04281=1108.656,5.283,-52.272,179.849,6.554,149.243
C04282=1108.661,5.033,-52.258,179.849,6.549,149.242
C04283=1108.666,4.785,-52.243,179.848,6.545,149.241
C04284=1108.671,4.535,-52.229,179.847,6.540,149.240
C04285=1108.676,4.286,-52.215,179.847,6.536,149.239
C04286=1108.681,4.037,-52.200,179.846,6.531,149.238
C04287=1108.687,3.787,-52.185,179.846,6.527,149.238
C04288=1108.691,3.537,-52.171,179.845,6.523,149.237
C04289=1108.696,3.287,-52.156,179.845,6.518,149.236
C04290=1108.701,3.038,-52.141,179.844,6.513,149.235
C04291=1108.706,2.788,-52.127,179.844,6.509,149.234
C04292=1108.711,2.539,-52.113,179.843,6.504,149.234
C04293=1108.716,2.289,-52.099,179.842,6.500,149.233
C04294=1108.721,2.040,-52.085,179.842,6.495,149.232
C04295=1108.727,1.791,-52.069,179.841,6.490,149.231
C04296=1108.732,1.541,-52.055,179.840,6.486,149.230
C04297=1108.737,1.291,-52.041,179.839,6.481,149.229
C04298=1108.742,1.041,-52.026,179.839,6.476,149.228
C04299=1108.747,0.792,-52.012,179.838,6.472,149.228
C04300=1108.752,0.542,-51.998,179.837,6.467,149.227
C04301=1108.757,0.294,-51.983,179.837,6.463,149.226
C04302=1108.762,0.044,-51.969,179.837,6.459,149.225
C04303=1108.767,-0.206,-51.954,179.836,6.454,149.224
C04304=1108.772,-0.456,-51.940,179.835,6.450,149.224
C04305=1108.777,-0.705,-51.926,179.835,6.445,149.223
C04306=1108.782,-0.955,-51.912,179.834,6.440,149.222
C04307=1108.787,-1.204,-51.898,179.833,6.436,149.221
C04308=1108.792,-1.454,-51.883,179.833,6.431,149.220
C04309=1108.797,-1.703,-51.869,179.832,6.426,149.219
C04310=1108.802,-1.953,-51.855,179.831,6.422,149.219
C04311=1108.807,-2.203,-51.841,179.831,6.417,149.218
C04312=1108.812,-2.451,-51.826,179.831,6.414,149.217
C04313=1108.817,-2.701,-51.812,179.830,6.409,149.216
C04314=1108.822,-2.951,-51.797,179.829,6.404,149.215
C04315=1108.827,-3.200,-51.783,179.829,6.400,149.214
C04316=1108.832,-3.450,-51.769,179.828,6.395,149.214
C04317=1108.837,-3.665,-51.758,179.828,6.392,149.213
C04318=1108.841,-3.879,-51.746,179.827,6.387,149.212
C04319=1108.845,-4.093,-51.733,179.827,6.384,149.212
C04320=1108.850,-4.307,-51.721,179.826,6.380,149.211
C04321=1108.855,-4.521,-51.709,179.826,6.375,149.210
C04322=1108.859,-4.736,-51.696,179.825,6.372,149.209
C04323=1108.863,-4.950,-51.684,179.825,6.368,149.209
C04324=1108.868,-5.164,-51.672,179.824,6.364,149.208
C04325=1108.873,-5.414,-51.658,179.823,6.359,149.207
C04326=1108.878,-5.664,-51.644,179.823,6.355,149.206
C04327=1108.882,-5.913,-51.631,179.822,6.351,149.206
C04328=1108.888,-6.162,-51.617,179.822,6.346,149.205
C04329=1108.893,-6.412,-51.602,179.821,6.342,149.204
C04330=1108.898,-6.662,-51.588,179.820,6.337,149.203
C04331=1108.903,-6.911,-51.574,179.820,6.333,149.202
C04332=1108.908,-7.160,-51.560,179.819,6.328,149.201
C04333=1108.913,-7.410,-51.546,179.819,6.323,149.200
C04334=1108.918,-7.660,-51.532,179.818,6.319,149.200
C04335=1108.923,-7.909,-51.519,179.817,6.314,149.199
C04336=1108.928,-8.159,-51.504,179.817,6.310,149.198
C04337=1108.933,-8.409,-51.490,179.817,6.305,149.197
C04338=1108.939,-8.658,-51.476,179.816,6.301,149.196
C04339=1108.944,-8.908,-51.463,179.815,6.296,149.195
C04340=1108.948,-9.157,-51.449,179.815,6.292,149.195
C04341=1108.953,-9.407,-51.435,179.814,6.287,149.194
C04342=1108.959,-9.656,-51.421,179.813,6.283,149.193
C04343=1108.964,-9.906,-51.407,179.813,6.278,149.192
C04344=1108.969,-10.156,-51.393,179.813,6.274,149.191
C04345=1108.974,-10.405,-51.380,179.813,6.269,149.190
C04346=1108.979,-10.654,-51.365,179.812,6.265,149.190
C04347=1108.984,-10.905,-51.352,179.811,6.260,149.189
C04348=1108.989,-11.154,-51.338,179.811,6.255,149.188
C04349=1108.994,-11.403,-51.324,179.810,6.251,149.187
C04350=1108.999,-11.652,-51.310,179.809,6.246,149.186
C04351=1109.004,-11.903,-51.297,179.809,6.242,149.185
C04352=1109.009,-12.152,-51.282,179.809,6.238,149.184
C04353=1109.014,-12.401,-51.269,179.808,6.233,149.184
C04354=1109.019,-12.651,-51.256,179.808,6.228,149.183
C04355=1109.024,-12.901,-51.241,179.807,6.224,149.182
C04356=1109.030,-13.150,-51.229,179.806,6.219,149.181
C04357=1109.034,-13.400,-51.214,179.806,6.214,149.180
C04358=1109.040,-13.649,-51.201,179.805,6.210,149.179
C04359=1109.045,-13.899,-51.188,179.805,6.205,149.178
C04360=1109.049,-14.149,-51.173,179.804,6.201,149.178
C04361=1109.055,-14.398,-51.159,179.804,6.197,149.177
C04362=1109.060,-14.648,-51.146,179.803,6.192,149.176
C04363=1109.065,-14.897,-51.133,179.803,6.187,149.175
C04364=1109.070,-15.147,-51.119,179.802,6.183,149.174
C04365=1109.075,-15.397,-51.105,179.802,6.178,149.173
C04366=1109.080,-15.646,-51.092,179.801,6.174,149.173
C04367=1109.085,-15.896,-51.078,179.800,6.169,149.172
C04368=1109.091,-16.145,-51.065,179.800,6.164,149.171
C04369=1109.096,-16.395,-51.051,179.800,6.160,149.170
C04370=1109.101,-16.645,-51.038,179.800,6.155,149.169
C04371=1109.106,-16.894,-51.024,179.799,6.151,149.168
C04372=1109.111,-17.144,-51.011,179.799,6.146,149.167
C04373=1109.115,-17.358,-50.998,179.798,6.142,149.167
C04374=1109.119,-17.572,-50.988,179.797,6.138,149.166
C04375=1109.124,-17.786,-50.976,179.797,6.134,149.165
C04376=1109.129,-18.001,-50.964,179.797,6.131,149.164
C04377=1109.133,-18.215,-50.953,179.796,6.126,149.164
C04378=1109.137,-18.430,-50.941,179.796,6.122,149.163
C04379=1109.141,-18.644,-50.930,179.796,6.119,149.162
C04380=1109.146,-18.858,-50.918,179.795,6.114,149.161
C04381=1109.152,-19.108,-50.905,179.795,6.109,149.160
C04382=1109.156,-19.358,-50.892,179.794,6.105,149.160
C04383=1109.162,-19.607,-50.878,179.793,6.100,149.159
C04384=1109.166,-19.857,-50.865,179.793,6.096,149.158
C04385=1109.172,-20.106,-50.851,179.793,6.092,149.157
C04386=1109.176,-20.356,-50.838,179.792,6.087,149.156
C04387=1109.182,-20.606,-50.825,179.792,6.082,149.155
C04388=1109.186,-20.855,-50.811,179.791,6.077,149.154
C04389=1109.192,-21.105,-50.798,179.791,6.073,149.153
C04390=1109.197,-21.355,-50.785,179.791,6.068,149.152
C04391=1109.202,-21.604,-50.771,179.790,6.063,149.151
C04392=1109.207,-21.854,-50.758,179.790,6.059,149.151
C04393=1109.213,-22.103,-50.745,179.789,6.054,149.150
C04394=1109.217,-22.353,-50.731,179.789,6.049,149.149
C04395=1109.223,-22.602,-50.718,179.789,6.045,149.148
C04396=1109.228,-22.852,-50.705,179.789,6.040,149.147
C04397=1109.233,-23.102,-50.692,179.788,6.035,149.146
C04398=1109.238,-23.351,-50.679,179.788,6.031,149.145
C04399=1109.242,-23.601,-50.666,179.787,6.026,149.144
C04400=1109.248,-23.850,-50.652,179.787,6.021,149.143
C04401=1109.253,-24.100,-50.639,179.786,6.016,149.142
C04402=1109.258,-24.349,-50.625,179.786,6.012,149.141
C04403=1109.264,-24.599,-50.613,179.785,6.007,149.140
C04404=1109.269,-24.849,-50.599,179.785,6.002,149.140
C04405=1109.274,-25.098,-50.587,179.785,5.997,149.138
C04406=1109.278,-25.348,-50.574,179.784,5.992,149.138
C04407=1109.284,-25.597,-50.560,179.784,5.988,149.137
C04408=1109.289,-25.847,-50.547,179.784,5.984,149.136
C04409=1109.294,-26.097,-50.534,179.784,5.979,149.135
C04410=1109.299,-26.346,-50.521,179.784,5.975,149.134
C04411=1109.304,-26.596,-50.508,179.784,5.970,149.133
C04412=1109.310,-26.846,-50.495,179.784,5.966,149.132
C04413=1109.315,-27.095,-50.482,179.784,5.961,149.131
C04414=1109.319,-27.345,-50.469,179.785,5.957,149.130
C04415=1109.325,-27.594,-50.455,179.784,5.952,149.129
C04416=1109.330,-27.844,-50.443,179.784,5.948,149.128
C04417=1109.335,-28.094,-50.430,179.784,5.943,149.127
C04418=1109.341,-28.343,-50.417,179.784,5.939,149.126
C04419=1109.346,-28.593,-50.404,179.784,5.934,149.125
C04420=1109.350,-28.843,-50.391,179.784,5.930,149.124
C04421=1109.355,-29.092,-50.379,179.784,5.925,149.123
C04422=1109.361,-29.342,-50.365,179.784,5.922,149.122
C04423=1109.366,-29.592,-50.352,179.783,5.917,149.121
C04424=1109.371,-29.841,-50.340,179.783,5.913,149.120
C04425=1109.376,-30.091,-50.326,179.783,5.908,149.119
C04426=1109.381,-30.341,-50.314,179.782,5.903,149.118
C04427=1109.386,-30.590,-50.301,179.783,5.899,149.118
C04428=1109.391,-30.840,-50.288,179.782,5.895,149.117
C04429=1109.396,-31.054,-50.277,179.782,5.891,149.116
C04430=1109.400,-31.269,-50.266,179.782,5.887,149.115
C04431=1109.404,-31.483,-50.255,179.782,5.883,149.114
C04432=1109.408,-31.697,-50.244,179.782,5.880,149.113
C04433=1109.413,-31.912,-50.233,179.781,5.876,149.113
C04434=1109.418,-32.127,-50.221,179.782,5.872,149.112
C04435=1109.422,-32.341,-50.211,179.781,5.869,149.111
C04436=1109.427,-32.555,-50.199,179.781,5.864,149.110
C04437=1109.432,-32.805,-50.187,179.781,5.860,149.109
C04438=1109.437,-33.054,-50.174,179.780,5.856,149.109
C04439=1109.442,-33.304,-50.161,179.779,5.851,149.108
C04440=1109.447,-33.553,-50.149,179.780,5.847,149.107
C04441=1109.453,-33.803,-50.135,179.779,5.842,149.106
C04442=1109.458,-34.052,-50.123,179.779,5.838,149.105
C04443=1109.462,-34.302,-50.110,179.779,5.834,149.104
C04444=1109.467,-34.552,-50.097,179.778,5.829,149.103
C04445=1109.473,-34.802,-50.085,179.777,5.825,149.103
C04446=1109.478,-35.051,-50.073,179.777,5.820,149.102
C04447=1109.483,-35.301,-50.059,179.777,5.815,149.101
C04448=1109.488,-35.551,-50.046,179.777,5.811,149.100
C04449=1109.493,-35.800,-50.034,179.776,5.806,149.099
C04450=1109.499,-36.049,-50.021,179.776,5.802,149.098
C04451=1109.503,-36.300,-50.009,179.775,5.797,149.097
C04452=1109.508,-36.549,-49.996,179.774,5.793,149.096
C04453=1109.514,-36.798,-49.984,179.774,5.788,149.096
C04454=1109.519,-37.048,-49.971,179.774,5.783,149.095
C04455=1109.524,-37.298,-49.958,179.773,5.778,149.094
C04456=1109.529,-37.548,-49.946,179.773,5.774,149.093
C04457=1109.535,-37.797,-49.933,179.772,5.769,149.092
C04458=1109.540,-38.047,-49.921,179.772,5.764,149.091
C04459=1109.545,-38.296,-49.908,179.771,5.760,149.090
C04460=1109.550,-38.546,-49.896,179.770,5.755,149.089
C04461=1109.555,-38.796,-49.883,179.770,5.750,149.089
C04462=1109.560,-39.045,-49.871,179.769,5.746,149.088
C04463=1109.565,-39.295,-49.858,179.769,5.741,149.087
C04464=1109.570,-39.545,-49.846,179.769,5.736,149.086
C04465=1109.576,-39.794,-49.833,179.768,5.731,149.085
C04466=1109.581,-40.043,-49.821,179.768,5.727,149.084
C04467=1109.586,-40.294,-49.808,179.767,5.722,149.083
C04468=1109.591,-40.543,-49.795,179.767,5.717,149.082
C04469=1109.596,-40.793,-49.783,179.766,5.712,149.081
C04470=1109.602,-41.043,-49.771,179.765,5.707,149.080
C04471=1109.607,-41.292,-49.758,179.765,5.702,149.079
C04472=1109.612,-41.541,-49.746,179.764,5.697,149.078
C04473=1109.618,-41.791,-49.734,179.763,5.692,149.078
C04474=1109.622,-42.041,-49.721,179.763,5.687,149.077
C04475=1109.628,-42.291,-49.709,179.763,5.682,149.076
C04476=1109.632,-42.540,-49.697,179.762,5.676,149.075
C04477=1109.637,-42.790,-49.685,179.762,5.672,149.074
C04478=1109.642,-43.039,-49.672,179.762,5.667,149.073
C04479=1109.648,-43.289,-49.660,179.761,5.662,149.072
C04480=1109.653,-43.539,-49.648,179.762,5.657,149.071
C04481=1109.658,-43.788,-49.635,179.762,5.652,149.069
C04482=1109.664,-44.038,-49.624,179.762,5.648,149.068
C04483=1109.669,-44.287,-49.611,179.762,5.643,149.067
C04484=1109.674,-44.538,-49.599,179.762,5.638,149.066
C04485=1109.678,-44.751,-49.588,179.762,5.634,149.065
C04486=1109.683,-44.966,-49.578,179.763,5.630,149.064
C04487=1109.687,-45.181,-49.567,179.763,5.626,149.063
C04488=1109.692,-45.396,-49.557,179.763,5.622,149.062
C04489=1109.696,-45.610,-49.546,179.763,5.618,149.062
C04490=1109.700,-45.825,-49.536,179.763,5.615,149.061
C04491=1109.705,-46.039,-49.525,179.763,5.611,149.060
C04492=1109.709,-46.254,-49.515,179.763,5.606,149.059
C04493=1109.714,-46.504,-49.502,179.764,5.602,149.058
C04494=1109.720,-46.754,-49.490,179.764,5.596,149.057
C04495=1109.724,-47.003,-49.478,179.764,5.592,149.055
C04496=1109.729,-47.252,-49.467,179.764,5.587,149.054
C04497=1109.735,-47.502,-49.454,179.764,5.582,149.053
C04498=1109.740,-47.752,-49.442,179.765,5.578,149.052
C04499=1109.745,-48.002,-49.430,179.764,5.573,149.051
C04500=1109.751,-48.251,-49.418,179.764,5.568,149.050
C04501=1109.756,-48.501,-49.406,179.765,5.564,149.049
C04502=1109.760,-48.750,-49.394,179.765,5.559,149.048
C04503=1109.766,-49.000,-49.382,179.765,5.555,149.047
C04504=1109.771,-49.250,-49.370,179.765,5.549,149.046
C04505=1109.776,-49.499,-49.357,179.765,5.544,149.045
C04506=1109.782,-49.749,-49.345,179.766,5.540,149.044
C04507=1109.787,-49.999,-49.334,179.766,5.535,149.043
C04508=1109.792,-50.248,-49.322,179.766,5.530,149.041
C04509=1109.797,-50.498,-49.310,179.766,5.526,149.040
C04510=1109.802,-50.748,-49.298,179.766,5.521,149.039
C04511=1109.808,-50.997,-49.285,179.767,5.517,149.038
C04512=1109.812,-51.247,-49.274,179.766,5.512,149.037
C04513=1109.818,-51.497,-49.262,179.766,5.507,149.036
C04514=1109.823,-51.746,-49.249,179.767,5.503,149.035
C04515=1109.828,-51.996,-49.238,179.767,5.497,149.034
C04516=1109.833,-52.246,-49.226,179.767,5.493,149.033
C04517=1109.838,-52.496,-49.214,179.767,5.488,149.032
C04518=1109.844,-52.745,-49.202,179.767,5.483,149.031
C04519=1109.849,-52.995,-49.190,179.768,5.479,149.030
C04520=1109.854,-53.244,-49.179,179.768,5.474,149.028
C04521=1109.860,-53.494,-49.167,179.768,5.469,149.027
C04522=1109.865,-53.743,-49.154,179.768,5.465,149.026
C04523=1109.869,-53.993,-49.143,179.768,5.460,149.025
C04524=1109.875,-54.243,-49.131,179.768,5.455,149.024
C04525=1109.880,-54.492,-49.119,179.768,5.451,149.023
C04526=1109.886,-54.742,-49.107,179.768,5.446,149.022
C04527=1109.890,-54.991,-49.095,179.768,5.441,149.021
C04528=1109.896,-55.241,-49.084,179.769,5.437,149.020
C04529=1109.901,-55.491,-49.072,179.769,5.432,149.019
C04530=1109.906,-55.741,-49.060,179.769,5.428,149.018
C04531=1109.911,-55.991,-49.049,179.769,5.422,149.017
C04532=1109.916,-56.240,-49.036,179.769,5.417,149.016
C04533=1109.921,-56.490,-49.025,179.769,5.413,149.015
C04534=1109.926,-56.740,-49.013,179.769,5.408,149.013
C04535=1109.932,-56.989,-49.002,179.769,5.403,149.013
C04536=1109.937,-57.239,-48.990,179.770,5.399,149.011
C04537=1109.943,-57.489,-48.978,179.770,5.394,149.010
C04538=1109.947,-57.738,-48.967,179.769,5.389,149.009
C04539=1109.953,-57.988,-48.955,179.770,5.385,149.008
C04540=1109.957,-58.237,-48.943,179.770,5.380,149.007
C04541=1109.961,-58.452,-48.933,179.770,5.376,149.006
C04542=1109.967,-58.666,-48.923,179.770,5.372,149.005
C04543=1109.971,-58.881,-48.913,179.770,5.368,149.004
C04544=1109.976,-59.096,-48.903,179.771,5.364,149.004
C04545=1109.980,-59.311,-48.893,179.771,5.360,149.003
C04546=1109.985,-59.525,-48.883,179.770,5.356,149.002
C04547=1109.989,-59.740,-48.873,179.771,5.352,149.001
C04548=1109.993,-59.954,-48.863,179.771,5.348,149.000
C04549=1109.998,-60.204,-48.851,179.770,5.343,148.999
C04550=1110.004,-60.454,-48.839,179.770,5.338,148.998
C04551=1110.008,-60.703,-48.828,179.770,5.333,148.997
C04552=1110.014,-60.953,-48.816,179.769,5.328,148.996
C04553=1110.019,-61.202,-48.805,179.769,5.323,148.995
C04554=1110.024,-61.452,-48.793,179.769,5.318,148.994
C04555=1110.029,-61.702,-48.782,179.768,5.313,148.993
C04556=1110.034,-61.952,-48.770,179.768,5.308,148.992
C04557=1110.040,-62.201,-48.759,179.767,5.303,148.991
C04558=1110.045,-62.451,-48.747,179.767,5.298,148.990
C04559=1110.050,-62.701,-48.737,179.767,5.293,148.989
C04560=1110.056,-62.951,-48.725,179.767,5.288,148.988
C04561=1110.060,-63.200,-48.713,179.767,5.283,148.987
C04562=1110.066,-63.450,-48.702,179.766,5.277,148.986
C04563=1110.071,-63.699,-48.691,179.766,5.272,148.985
C04564=1110.076,-63.949,-48.679,179.765,5.267,148.984
C04565=1110.081,-64.199,-48.667,179.765,5.262,148.983
C04566=1110.087,-64.449,-48.656,179.765,5.258,148.982
C04567=1110.092,-64.698,-48.645,179.765,5.252,148.981
C04568=1110.098,-64.948,-48.633,179.764,5.247,148.980
C04569=1110.102,-65.198,-48.622,179.764,5.242,148.979
C04570=1110.107,-65.448,-48.611,179.764,5.237,148.978
C04571=1110.113,-65.697,-48.599,179.764,5.232,148.976
C04572=1110.118,-65.946,-48.588,179.764,5.227,148.976
C04573=1110.123,-66.196,-48.576,179.764,5.222,148.974
C04574=1110.128,-66.447,-48.566,179.763,5.216,148.973
C04575=1110.133,-66.696,-48.555,179.763,5.211,148.972
C04576=1110.139,-66.945,-48.543,179.763,5.206,148.971
C04577=1110.144,-67.195,-48.531,179.763,5.201,148.970
C04578=1110.149,-67.446,-48.520,179.763,5.196,148.969
C04579=1110.155,-67.695,-48.509,179.762,5.191,148.968
C04580=1110.159,-67.944,-48.498,179.762,5.186,148.967
C04581=1110.165,-68.194,-48.486,179.762,5.180,148.966
C04582=1110.170,-68.444,-48.476,179.762,5.176,148.965
C04583=1110.175,-68.693,-48.465,179.762,5.170,148.964
C04584=1110.180,-68.943,-48.453,179.762,5.165,148.962
C04585=1110.186,-69.192,-48.442,179.762,5.160,148.961
C04586=1110.191,-69.442,-48.431,179.762,5.155,148.960
C04587=1110.196,-69.692,-48.419,179.762,5.150,148.959
C04588=1110.201,-69.941,-48.409,179.761,5.144,148.958
C04589=1110.206,-70.192,-48.398,179.761,5.140,148.957
C04590=1110.212,-70.441,-48.386,179.761,5.134,148.956
C04591=1110.217,-70.690,-48.375,179.761,5.129,148.955
C04592=1110.222,-70.941,-48.365,179.761,5.124,148.954
C04593=1110.227,-71.190,-48.353,179.762,5.119,148.952
C04594=1110.233,-71.440,-48.342,179.761,5.114,148.952
C04595=1110.238,-71.690,-48.331,179.761,5.109,148.950
C04596=1110.243,-71.939,-48.320,179.761,5.104,148.949
C04597=1110.248,-72.154,-48.311,179.761,5.099,148.948
C04598=1110.252,-72.369,-48.301,179.761,5.094,148.947
C04599=1110.257,-72.583,-48.291,179.761,5.090,148.946
C04600=1110.261,-72.798,-48.283,179.761,5.085,148.945
C04601=1110.265,-73.013,-48.273,179.761,5.081,148.944
C04602=1110.270,-73.227,-48.263,179.761,5.077,148.943
C04603=1110.274,-73.443,-48.254,179.761,5.073,148.942
C04604=1110.279,-73.657,-48.245,179.761,5.068,148.942
C04605=1110.284,-73.907,-48.234,179.761,5.063,148.940
C04606=1110.290,-74.156,-48.223,179.761,5.058,148.939
C04607=1110.295,-74.406,-48.212,179.761,5.053,148.938
C04608=1110.300,-74.656,-48.201,179.761,5.047,148.937
C04609=1110.305,-74.906,-48.190,179.762,5.042,148.936
C04610=1110.310,-75.155,-48.179,179.762,5.037,148.934
C04611=1110.316,-75.405,-48.168,179.762,5.032,148.933
C04612=1110.321,-75.655,-48.157,179.762,5.027,148.932
C04613=1110.327,-75.904,-48.147,179.762,5.022,148.931
C04614=1110.331,-76.154,-48.136,179.762,5.017,148.930
C04615=1110.336,-76.404,-48.125,179.762,5.011,148.929
C04616=1110.342,-76.653,-48.114,179.763,5.006,148.927
C04617=1110.347,-76.904,-48.103,179.763,5.001,148.926
C04618=1110.353,-77.153,-48.093,179.763,4.996,148.925
C04619=1110.358,-77.403,-48.081,179.763,4.991,148.924
C04620=1110.363,-77.652,-48.071,179.763,4.986,148.923
C04621=1110.368,-77.902,-48.060,179.763,4.981,148.922
C04622=1110.374,-78.151,-48.050,179.764,4.975,148.920
C04623=1110.379,-78.402,-48.039,179.764,4.970,148.919
C04624=1110.384,-78.651,-48.028,179.764,4.965,148.918
C04625=1110.390,-78.901,-48.017,179.764,4.960,148.917
C04626=1110.395,-79.151,-48.007,179.764,4.955,148.916
C04627=1110.400,-79.400,-47.996,179.764,4.950,148.915
C04628=1110.406,-79.650,-47.985,179.764,4.944,148.913
C04629=1110.411,-79.900,-47.975,179.765,4.939,148.912
C04630=1110.416,-80.149,-47.964,179.765,4.934,148.911
C04631=1110.421,-80.399,-47.953,179.765,4.929,148.910
C04632=1110.426,-80.649,-47.943,179.765,4.924,148.909
C04633=1110.431,-80.898,-47.932,179.765,4.919,148.907
C04634=1110.437,-81.148,-47.922,179.765,4.914,148.906
C04635=1110.442,-81.398,-47.911,179.766,4.908,148.905
C04636=1110.447,-81.648,-47.901,179.766,4.903,148.904
C04637=1110.452,-81.897,-47.889,179.767,4.899,148.903
C04638=1110.458,-82.147,-47.879,179.767,4.893,148.901
C04639=1110.463,-82.397,-47.869,179.767,4.888,148.900
C04640=1110.468,-82.647,-47.858,179.768,4.883,148.899
C04641=1110.473,-82.896,-47.847,179.768,4.878,148.898
C04642=1110.479,-83.146,-47.837,179.768,4.873,148.897
C04643=1110.484,-83.395,-47.827,179.768,4.868,148.895
C04644=1110.489,-83.646,-47.816,179.768,4.863,148.894
C04645=1110.495,-83.895,-47.806,179.768,4.857,148.893
C04646=1110.499,-84.145,-47.795,179.770,4.853,148.892
C04647=1110.505,-84.394,-47.785,179.770,4.848,148.891
C04648=1110.510,-84.645,-47.774,179.770,4.842,148.889
C04649=1110.516,-84.894,-47.764,179.770,4.837,148.888
C04650=1110.521,-85.144,-47.753,179.770,4.832,148.887
C04651=1110.526,-85.394,-47.743,179.771,4.827,148.886
C04652=1110.531,-85.643,-47.732,179.771,4.823,148.885
C04653=1110.535,-85.858,-47.723,179.772,4.817,148.883
C04654=1110.541,-86.073,-47.714,179.772,4.814,148.882
C04655=1110.545,-86.288,-47.706,179.772,4.810,148.882
C04656=1110.549,-86.502,-47.696,179.772,4.804,148.880
C04657=1110.553,-86.717,-47.687,179.772,4.800,148.879
C04658=1110.559,-86.932,-47.678,179.773,4.796,148.878
C04659=1110.563,-87.147,-47.670,179.774,4.792,148.877
C04660=1110.568,-87.362,-47.661,179.773,4.787,148.876
C04661=1110.572,-87.611,-47.650,179.774,4.783,148.875
C04662=1110.577,-87.861,-47.640,179.775,4.778,148.874
C04663=1110.583,-88.111,-47.630,179.775,4.772,148.873
C04664=1110.589,-88.360,-47.620,179.775,4.767,148.871
C04665=1110.594,-88.610,-47.609,179.776,4.763,148.870
C04666=1110.599,-88.860,-47.599,179.776,4.758,148.869
C04667=1110.604,-89.110,-47.588,179.776,4.753,148.868
C04668=1110.610,-89.360,-47.578,179.777,4.748,148.866
C04669=1110.615,-89.609,-47.568,179.778,4.743,148.865
C04670=1110.620,-89.859,-47.558,179.778,4.738,148.864
C04671=1110.625,-90.109,-47.548,179.778,4.732,148.863
C04672=1110.631,-90.358,-47.537,179.779,4.728,148.862
C04673=1110.636,-90.608,-47.527,179.779,4.723,148.860
C04674=1110.641,-90.858,-47.517,179.779,4.718,148.859
C04675=1110.646,-91.107,-47.507,179.780,4.713,148.858
C04676=1110.651,-91.357,-47.496,179.781,4.708,148.857
C04677=1110.657,-91.607,-47.486,179.781,4.703,148.855
C04678=1110.662,-91.857,-47.476,179.782,4.698,148.854
C04679=1110.667,-92.107,-47.465,179.782,4.693,148.853
C04680=1110.672,-92.356,-47.456,179.783,4.689,148.852
C04681=1110.678,-92.606,-47.446,179.783,4.684,148.851
C04682=1110.683,-92.856,-47.435,179.783,4.679,148.850
C04683=1110.688,-93.105,-47.425,179.784,4.674,148.848
C04684=1110.694,-93.356,-47.415,179.784,4.669,148.847
C04685=1110.699,-93.605,-47.405,179.785,4.665,148.846
C04686=1110.704,-93.855,-47.395,179.786,4.659,148.845
C04687=1110.710,-94.105,-47.385,179.786,4.654,148.843
C04688=1110.715,-94.354,-47.375,179.787,4.650,148.842
C04689=1110.720,-94.604,-47.365,179.787,4.645,148.841
C04690=1110.725,-94.854,-47.354,179.787,4.639,148.840
C04691=1110.731,-95.103,-47.344,179.788,4.635,148.839
C04692=1110.736,-95.353,-47.334,179.788,4.630,148.837
C04693=1110.741,-95.603,-47.325,179.788,4.625,148.836
C04694=1110.747,-95.853,-47.315,179.788,4.621,148.835
C04695=1110.752,-96.102,-47.304,179.789,4.616,148.834
C04696=1110.757,-96.352,-47.294,179.789,4.611,148.833
C04697=1110.762,-96.602,-47.284,179.789,4.605,148.832
C04698=1110.768,-96.851,-47.274,179.790,4.601,148.831
C04699=1110.774,-97.101,-47.264,179.790,4.596,148.829
C04700=1110.778,-97.351,-47.255,179.790,4.591,148.828
C04701=1110.783,-97.601,-47.244,179.791,4.586,148.827
C04702=1110.789,-97.851,-47.234,179.791,4.581,148.826
C04703=1110.794,-98.100,-47.224,179.791,4.576,148.825
C04704=1110.799,-98.351,-47.215,179.792,4.571,148.823
C04705=1110.805,-98.600,-47.204,179.792,4.567,148.822
C04706=1110.810,-98.849,-47.195,179.793,4.561,148.821
C04707=1110.815,-99.099,-47.185,179.793,4.556,148.820
C04708=1110.821,-99.349,-47.175,179.793,4.551,148.819
C04709=1110.825,-99.564,-47.166,179.794,4.547,148.817
C04710=1110.830,-99.779,-47.158,179.794,4.543,148.816
C04711=1110.834,-99.993,-47.150,179.795,4.539,148.815
C04712=1110.839,-100.209,-47.140,179.795,4.535,148.815
C04713=1110.843,-100.423,-47.132,179.795,4.530,148.813
C04714=1110.848,-100.638,-47.125,179.795,4.526,148.812
C04715=1110.852,-100.853,-47.116,179.796,4.522,148.811
C04716=1110.857,-101.068,-47.107,179.796,4.517,148.810
C04717=1110.862,-101.317,-47.097,179.797,4.512,148.809
C04718=1110.868,-101.568,-47.088,179.797,4.507,148.808
C04719=1110.874,-101.817,-47.078,179.797,4.502,148.807
C04720=1110.878,-102.067,-47.068,179.798,4.498,148.805
C04721=1110.884,-102.317,-47.058,179.798,4.493,148.804
C04722=1110.889,-102.566,-47.048,179.798,4.487,148.803
C04723=1110.894,-102.816,-47.038,179.799,4.482,148.802
C04724=1110.899,-103.066,-47.029,179.799,4.477,148.801
C04725=1110.904,-103.316,-47.019,179.800,4.473,148.799
C04726=1110.909,-103.565,-47.009,179.800,4.468,148.798
C04727=1110.915,-103.816,-47.000,179.800,4.462,148.797
C04728=1110.921,-104.065,-46.989,179.800,4.457,148.796
C04729=1110.926,-104.315,-46.981,179.801,4.453,148.795
C04730=1110.932,-104.564,-46.970,179.801,4.448,148.793
C04731=1110.936,-104.814,-46.961,179.802,4.443,148.792
C04732=1110.942,-105.065,-46.951,179.802,4.437,148.791
C04733=1110.947,-105.314,-46.941,179.802,4.432,148.790
C04734=1110.952,-105.564,-46.932,179.803,4.428,148.789
C04735=1110.957,-105.813,-46.922,179.803,4.423,148.787
C04736=1110.963,-106.063,-46.913,179.803,4.418,148.786
C04737=1110.968,-106.313,-46.903,179.804,4.412,148.785
C04738=1110.974,-106.563,-46.894,179.804,4.407,148.784
C04739=1110.978,-106.813,-46.884,179.804,4.402,148.783
C04740=1110.984,-107.063,-46.874,179.805,4.398,148.781
C04741=1110.989,-107.312,-46.865,179.805,4.393,148.780
C04742=1110.995,-107.562,-46.855,179.805,4.387,148.779
C04743=1111.000,-107.811,-46.845,179.806,4.382,148.778
C04744=1111.005,-108.061,-46.837,179.806,4.377,148.777
C04745=1111.011,-108.311,-46.826,179.806,4.372,148.775
C04746=1111.016,-108.561,-46.817,179.807,4.368,148.774
C04747=1111.021,-108.810,-46.807,179.807,4.362,148.773
C04748=1111.026,-109.060,-46.798,179.808,4.357,148.772
C04749=1111.032,-109.310,-46.788,179.808,4.352,148.770
C04750=1111.037,-109.559,-46.779,179.809,4.347,148.769
C04751=1111.042,-109.810,-46.769,179.809,4.341,148.768
C04752=1111.047,-110.060,-46.760,179.810,4.337,148.767
C04753=1111.053,-110.309,-46.751,179.810,4.332,148.766
C04754=1111.058,-110.559,-46.741,179.810,4.327,148.764
C04755=1111.063,-110.809,-46.732,179.810,4.322,148.763
C04756=1111.069,-111.058,-46.721,179.811,4.316,148.762
C04757=1111.074,-111.308,-46.713,179.811,4.311,148.761
C04758=1111.079,-111.558,-46.704,179.811,4.306,148.760
C04759=1111.085,-111.808,-46.693,179.812,4.301,148.758
C04760=1111.090,-112.057,-46.685,179.813,4.296,148.757
C04761=1111.095,-112.307,-46.676,179.813,4.291,148.756
C04762=1111.101,-112.557,-46.665,179.813,4.286,148.754
C04763=1111.106,-112.807,-46.657,179.813,4.281,148.753
C04764=1111.111,-113.057,-46.648,179.814,4.276,148.752
C04765=1111.116,-113.271,-46.639,179.814,4.272,148.751
C04766=1111.121,-113.486,-46.631,179.814,4.267,148.750
C04767=1111.125,-113.702,-46.622,179.815,4.263,148.749
C04768=1111.130,-113.917,-46.615,179.815,4.257,148.748
C04769=1111.134,-114.131,-46.607,179.815,4.253,148.747
C04770=1111.139,-114.346,-46.599,179.816,4.249,148.746
C04771=1111.144,-114.561,-46.591,179.816,4.244,148.745
C04772=1111.149,-114.776,-46.583,179.816,4.240,148.744
C04773=1111.154,-115.026,-46.574,179.817,4.235,148.742
C04774=1111.159,-115.275,-46.564,179.817,4.230,148.741
C04775=1111.164,-115.525,-46.555,179.817,4.224,148.740
C04776=1111.170,-115.775,-46.546,179.818,4.219,148.739
C04777=1111.175,-116.025,-46.537,179.818,4.214,148.737
C04778=1111.180,-116.275,-46.528,179.818,4.209,148.736
C04779=1111.186,-116.524,-46.518,179.819,4.203,148.735
C04780=1111.191,-116.774,-46.509,179.819,4.198,148.733
C04781=1111.196,-117.024,-46.500,179.820,4.193,148.732
C04782=1111.201,-117.274,-46.491,179.820,4.189,148.731
C04783=1111.207,-117.524,-46.482,179.821,4.184,148.730
C04784=1111.212,-117.773,-46.472,179.822,4.178,148.728
C04785=1111.217,-118.023,-46.463,179.822,4.173,148.727
C04786=1111.222,-118.273,-46.454,179.822,4.168,148.726
C04787=1111.228,-118.523,-46.445,179.822,4.163,148.725
C04788=1111.233,-118.773,-46.436,179.823,4.157,148.723
C04789=1111.238,-119.023,-46.427,179.823,4.152,148.722
C04790=1111.244,-119.271,-46.418,179.824,4.147,148.721
C04791=1111.250,-119.521,-46.408,179.824,4.142,148.720
C04792=1111.255,-119.771,-46.400,179.824,4.136,148.718
C04793=1111.260,-120.021,-46.391,179.825,4.131,148.717
C04794=1111.265,-120.271,-46.382,179.825,4.126,148.716
C04795=1111.270,-120.521,-46.373,179.826,4.121,148.715
C04796=1111.276,-120.771,-46.364,179.826,4.115,148.713
C04797=1111.282,-121.021,-46.354,179.827,4.110,148.712
C04798=1111.287,-121.271,-46.346,179.827,4.105,148.711
C04799=1111.292,-121.520,-46.337,179.827,4.099,148.709
C04800=1111.298,-121.770,-46.328,179.828,4.094,148.708
C04801=1111.303,-122.019,-46.319,179.828,4.088,148.707
C04802=1111.308,-122.269,-46.310,179.828,4.083,148.706
C04803=1111.313,-122.519,-46.301,179.829,4.077,148.704
C04804=1111.319,-122.769,-46.291,179.829,4.072,148.703
C04805=1111.324,-123.019,-46.282,179.829,4.067,148.702
C04806=1111.329,-123.268,-46.273,179.830,4.062,148.700
C04807=1111.334,-123.518,-46.265,179.831,4.056,148.699
C04808=1111.340,-123.767,-46.256,179.831,4.051,148.698
C04809=1111.345,-124.017,-46.247,179.831,4.046,148.696
C04810=1111.351,-124.268,-46.239,179.832,4.040,148.695
C04811=1111.356,-124.518,-46.230,179.832,4.035,148.694
C04812=1111.361,-124.767,-46.221,179.833,4.030,148.692
C04813=1111.367,-125.018,-46.212,179.833,4.024,148.691
C04814=1111.373,-125.267,-46.203,179.834,4.019,148.690
C04815=1111.378,-125.517,-46.194,179.834,4.013,148.688
C04816=1111.383,-125.766,-46.185,179.834,4.008,148.687
C04817=1111.388,-126.016,-46.176,179.835,4.003,148.686
C04818=1111.393,-126.266,-46.167,179.835,3.997,148.685
C04819=1111.399,-126.515,-46.159,179.836,3.992,148.683
C04820=1111.404,-126.765,-46.150,179.836,3.986,148.682
C04821=1111.409,-126.980,-46.142,179.836,3.982,148.681
C04822=1111.413,-127.195,-46.135,179.837,3.977,148.680
C04823=1111.418,-127.410,-46.128,179.837,3.972,148.678
C04824=1111.423,-127.625,-46.120,179.838,3.968,148.677
C04825=1111.428,-127.840,-46.113,179.838,3.963,148.676
C04826=1111.432,-128.055,-46.106,179.838,3.958,148.675
C04827=1111.436,-128.271,-46.098,179.839,3.954,148.674
C04828=1111.441,-128.486,-46.090,179.839,3.949,148.673
C04829=1111.018,-128.476,-46.116,179.847,3.953,148.671
C04830=1111.013,-128.261,-46.123,179.846,3.958,148.673
C04831=1111.008,-128.046,-46.131,179.846,3.962,148.674
C04832=1111.004,-127.832,-46.139,179.845,3.968,148.675
C04833=1110.999,-127.617,-46.146,179.845,3.972,148.676
C04834=1110.995,-127.402,-46.154,179.845,3.977,148.677
C04835=1110.990,-127.187,-46.161,179.844,3.981,148.678
C04836=1110.986,-126.971,-46.169,179.844,3.986,148.679
C04837=1110.982,-126.756,-46.176,179.843,3.990,148.681
C04838=1110.976,-126.507,-46.185,179.843,3.996,148.682
C04839=1110.971,-126.257,-46.194,179.843,4.002,148.683
C04840=1110.965,-126.007,-46.203,179.842,4.007,148.685
C04841=1110.960,-125.757,-46.212,179.841,4.012,148.686
C04842=1110.954,-125.507,-46.221,179.841,4.018,148.687
C04843=1110.949,-125.258,-46.230,179.841,4.023,148.688
C04844=1110.943,-125.008,-46.239,179.840,4.028,148.690
C04845=1110.938,-124.758,-46.247,179.840,4.033,148.691
C04846=1110.933,-124.508,-46.256,179.839,4.039,148.692
C04847=1110.928,-124.258,-46.265,179.839,4.044,148.694
C04848=1110.922,-124.008,-46.273,179.839,4.050,148.695
C04849=1110.917,-123.758,-46.282,179.838,4.056,148.696
C04850=1110.912,-123.509,-46.291,179.838,4.061,148.698
C04851=1110.906,-123.260,-46.301,179.837,4.066,148.699
C04852=1110.901,-123.010,-46.310,179.837,4.072,148.700
C04853=1110.896,-122.760,-46.319,179.836,4.077,148.702
C04854=1110.890,-122.510,-46.328,179.836,4.082,148.703
C04855=1110.885,-122.260,-46.337,179.835,4.087,148.704
C04856=1110.880,-122.010,-46.346,179.835,4.093,148.705
C04857=1110.875,-121.760,-46.354,179.835,4.098,148.707
C04858=1110.868,-121.511,-46.364,179.834,4.103,148.708
C04859=1110.863,-121.261,-46.372,179.834,4.108,148.709
C04860=1110.858,-121.011,-46.381,179.833,4.114,148.711
C04861=1110.853,-120.761,-46.390,179.833,4.119,148.712
C04862=1110.848,-120.512,-46.399,179.832,4.124,148.713
C04863=1110.842,-120.261,-46.409,179.832,4.129,148.714
C04864=1110.837,-120.012,-46.418,179.832,4.135,148.716
C04865=1110.832,-119.762,-46.427,179.831,4.140,148.717
C04866=1110.827,-119.512,-46.436,179.831,4.145,148.718
C04867=1110.822,-119.263,-46.445,179.830,4.151,148.720
C04868=1110.816,-119.012,-46.454,179.830,4.156,148.721
C04869=1110.810,-118.763,-46.463,179.830,4.161,148.722
C04870=1110.805,-118.513,-46.472,179.829,4.166,148.723
C04871=1110.800,-118.264,-46.481,179.829,4.172,148.725
C04872=1110.794,-118.014,-46.491,179.828,4.177,148.726
C04873=1110.789,-117.764,-46.500,179.828,4.182,148.727
C04874=1110.784,-117.514,-46.509,179.828,4.187,148.728
C04875=1110.778,-117.264,-46.518,179.827,4.193,148.730
C04876=1110.773,-117.015,-46.528,179.827,4.198,148.731
C04877=1110.768,-116.765,-46.537,179.827,4.203,148.732
C04878=1110.762,-116.515,-46.546,179.826,4.208,148.733
C04879=1110.757,-116.265,-46.555,179.826,4.213,148.735
C04880=1110.752,-116.016,-46.565,179.825,4.219,148.736
C04881=1110.747,-115.766,-46.574,179.825,4.224,148.737
C04882=1110.741,-115.516,-46.583,179.824,4.228,148.738
C04883=1110.735,-115.266,-46.592,179.824,4.233,148.740
C04884=1110.731,-115.017,-46.602,179.824,4.239,148.741
C04885=1110.725,-114.767,-46.611,179.823,4.244,148.742
C04886=1110.721,-114.552,-46.618,179.823,4.249,148.743
C04887=1110.716,-114.337,-46.627,179.823,4.253,148.744
C04888=1110.712,-114.122,-46.635,179.822,4.257,148.745
C04889=1110.707,-113.907,-46.643,179.822,4.262,148.746
C04890=1110.702,-113.692,-46.651,179.821,4.266,148.748
C04891=1110.697,-113.477,-46.659,179.821,4.270,148.749
C04892=1110.693,-113.262,-46.667,179.821,4.275,148.750
C04893=1110.688,-113.048,-46.675,179.820,4.279,148.751
C04894=1110.683,-112.798,-46.684,179.820,4.285,148.752
C04895=1110.678,-112.549,-46.694,179.820,4.290,148.753
C04896=1110.672,-112.298,-46.703,179.820,4.295,148.754
C04897=1110.668,-112.048,-46.713,179.819,4.300,148.756
C04898=1110.662,-111.798,-46.723,179.819,4.305,148.757
C04899=1110.657,-111.548,-46.732,179.818,4.310,148.758
C04900=1110.652,-111.299,-46.741,179.817,4.315,148.760
C04901=1110.646,-111.049,-46.751,179.817,4.320,148.761
C04902=1110.641,-110.799,-46.760,179.817,4.325,148.762
C04903=1110.635,-110.550,-46.770,179.817,4.331,148.763
C04904=1110.630,-110.300,-46.779,179.816,4.336,148.764
C04905=1110.625,-110.051,-46.788,179.816,4.341,148.766
C04906=1110.619,-109.800,-46.798,179.816,4.346,148.767
C04907=1110.614,-109.551,-46.808,179.815,4.350,148.768
C04908=1110.609,-109.301,-46.817,179.815,4.356,148.769
C04909=1110.603,-109.051,-46.826,179.815,4.361,148.770
C04910=1110.598,-108.802,-46.836,179.814,4.366,148.772
C04911=1110.593,-108.552,-46.845,179.814,4.371,148.773
C04912=1110.588,-108.302,-46.856,179.813,4.377,148.774
C04913=1110.582,-108.052,-46.864,179.813,4.381,148.775
C04914=1110.578,-107.802,-46.874,179.812,4.386,148.777
C04915=1110.572,-107.552,-46.884,179.812,4.391,148.778
C04916=1110.567,-107.303,-46.893,179.812,4.396,148.779
C04917=1110.561,-107.053,-46.903,179.812,4.402,148.780
C04918=1110.556,-106.804,-46.912,179.811,4.407,148.781
C04919=1110.550,-106.554,-46.923,179.811,4.411,148.783
C04920=1110.546,-106.304,-46.932,179.810,4.416,148.784
C04921=1110.540,-106.054,-46.942,179.810,4.421,148.785
C04922=1110.535,-105.804,-46.951,179.810,4.427,148.786
C04923=1110.530,-105.555,-46.961,179.810,4.432,148.787
C04924=1110.524,-105.304,-46.971,179.809,4.436,148.789
C04925=1110.519,-105.055,-46.980,179.809,4.441,148.790
C04926=1110.513,-104.806,-46.990,179.808,4.446,148.791
C04927=1110.509,-104.555,-47.000,179.808,4.452,148.792
C04928=1110.503,-104.306,-47.010,179.808,4.457,148.793
C04929=1110.498,-104.056,-47.019,179.807,4.461,148.795
C04930=1110.492,-103.806,-47.029,179.807,4.466,148.796
C04931=1110.487,-103.557,-47.039,179.807,4.471,148.797
C04932=1110.481,-103.307,-47.048,179.806,4.476,148.798
C04933=1110.477,-103.057,-47.058,179.805,4.481,148.799
C04934=1110.472,-102.807,-47.068,179.805,4.486,148.801
C04935=1110.466,-102.557,-47.078,179.805,4.491,148.802
C04936=1110.461,-102.308,-47.087,179.804,4.497,148.803
C04937=1110.455,-102.058,-47.098,179.804,4.502,148.804
C04938=1110.451,-101.808,-47.107,179.803,4.506,148.806
C04939=1110.445,-101.558,-47.117,179.803,4.511,148.807
C04940=1110.439,-101.309,-47.127,179.803,4.516,148.808
C04941=1110.434,-101.059,-47.136,179.803,4.522,148.809
C04942=1110.429,-100.844,-47.145,179.802,4.526,148.810
C04943=1110.425,-100.629,-47.154,179.802,4.530,148.811
C04944=1110.421,-100.414,-47.162,179.802,4.534,148.812
C04945=1110.416,-100.200,-47.170,179.801,4.538,148.813
C04946=1110.412,-99.984,-47.180,179.801,4.543,148.814
C04947=1110.407,-99.770,-47.188,179.801,4.547,148.815
C04948=1110.402,-99.556,-47.196,179.800,4.551,148.816
C04949=1110.399,-99.340,-47.205,179.800,4.555,148.817
C04950=1110.393,-99.090,-47.215,179.800,4.560,148.819
C04951=1110.387,-98.841,-47.225,179.799,4.565,148.820
C04952=1110.382,-98.591,-47.234,179.799,4.570,148.821
C04953=1110.377,-98.342,-47.245,179.798,4.575,148.822
C04954=1110.371,-98.091,-47.254,179.798,4.580,148.823
C04955=1110.366,-97.842,-47.264,179.798,4.585,148.825
C04956=1110.361,-97.592,-47.274,179.798,4.590,148.826
C04957=1110.355,-97.343,-47.285,179.797,4.595,148.827
C04958=1110.350,-97.092,-47.295,179.797,4.600,148.828
C04959=1110.345,-96.843,-47.305,179.796,4.605,148.829
C04960=1110.340,-96.593,-47.314,179.796,4.609,148.830
C04961=1110.335,-96.343,-47.325,179.795,4.614,148.832
C04962=1110.330,-96.094,-47.334,179.795,4.619,148.833
C04963=1110.324,-95.844,-47.345,179.795,4.625,148.834
C04964=1110.318,-95.595,-47.355,179.794,4.629,148.835
C04965=1110.313,-95.344,-47.365,179.794,4.634,148.836
C04966=1110.309,-95.095,-47.375,179.794,4.639,148.838
C04967=1110.303,-94.845,-47.384,179.793,4.644,148.839
C04968=1110.298,-94.595,-47.395,179.793,4.649,148.840
C04969=1110.292,-94.345,-47.405,179.793,4.654,148.841
C04970=1110.286,-94.096,-47.415,179.792,4.658,148.842
C04971=1110.282,-93.846,-47.425,179.792,4.663,148.844
C04972=1110.277,-93.596,-47.436,179.791,4.669,148.845
C04973=1110.271,-93.347,-47.446,179.791,4.673,148.846
C04974=1110.265,-93.097,-47.456,179.790,4.678,148.847
C04975=1110.261,-92.847,-47.466,179.790,4.682,148.848
C04976=1110.256,-92.598,-47.476,179.789,4.688,148.850
C04977=1110.250,-92.348,-47.486,179.789,4.693,148.851
C04978=1110.245,-92.098,-47.497,179.788,4.697,148.852
C04979=1110.239,-91.848,-47.507,179.788,4.702,148.853
C04980=1110.234,-91.599,-47.517,179.787,4.707,148.855
C04981=1110.230,-91.349,-47.527,179.787,4.712,148.856
C04982=1110.224,-91.099,-47.538,179.787,4.717,148.857
C04983=1110.218,-90.850,-47.548,179.786,4.722,148.858
C04984=1110.213,-90.599,-47.558,179.786,4.727,148.859
C04985=1110.208,-90.350,-47.569,179.785,4.732,148.860
C04986=1110.203,-90.100,-47.579,179.785,4.736,148.862
C04987=1110.198,-89.850,-47.589,179.784,4.741,148.863
C04988=1110.192,-89.601,-47.599,179.784,4.746,148.864
C04989=1110.187,-89.351,-47.610,179.784,4.752,148.865
C04990=1110.182,-89.101,-47.620,179.783,4.756,148.867
C04991=1110.176,-88.851,-47.630,179.783,4.761,148.868
C04992=1110.171,-88.601,-47.641,179.782,4.767,148.869
C04993=1110.165,-88.352,-47.651,179.782,4.771,148.870
C04994=1110.160,-88.101,-47.661,179.781,4.776,148.871
C04995=1110.156,-87.852,-47.671,179.781,4.781,148.873
C04996=1110.150,-87.603,-47.681,179.781,4.786,148.874
C04997=1110.145,-87.353,-47.693,179.780,4.792,148.875
C04998=1110.140,-87.138,-47.701,179.780,4.796,148.876
C04999=1110.136,-86.923,-47.710,179.780,4.800,148.877
C05000=1110.131,-86.708,-47.719,179.779,4.804,148.878
C05001=1110.127,-86.494,-47.728,179.779,4.809,148.879
C05002=1110.122,-86.279,-47.737,179.779,4.813,148.880
C05003=1110.118,-86.065,-47.746,179.778,4.817,148.881
C05004=1110.113,-85.849,-47.755,179.778,4.821,148.882
C05005=1110.109,-85.635,-47.764,179.778,4.826,148.883
C05006=1110.104,-85.385,-47.775,179.777,4.831,148.885
C05007=1110.098,-85.135,-47.785,179.777,4.836,148.886
C05008=1110.093,-84.885,-47.795,179.777,4.841,148.887
C05009=1110.088,-84.636,-47.806,179.777,4.846,148.888
C05010=1110.082,-84.387,-47.817,179.776,4.851,148.889
C05011=1110.077,-84.136,-47.827,179.776,4.857,148.891
C05012=1110.072,-83.887,-47.837,179.776,4.862,148.892
C05013=1110.067,-83.637,-47.848,179.775,4.866,148.893
C05014=1110.061,-83.388,-47.859,179.775,4.871,148.894
C05015=1110.056,-83.137,-47.869,179.775,4.877,148.895
C05016=1110.051,-82.888,-47.880,179.774,4.882,148.897
C05017=1110.046,-82.638,-47.890,179.774,4.887,148.898
C05018=1110.040,-82.389,-47.901,179.774,4.892,148.899
C05019=1110.035,-82.139,-47.912,179.774,4.897,148.900
C05020=1110.030,-81.889,-47.922,179.774,4.902,148.901
C05021=1110.025,-81.639,-47.932,179.773,4.908,148.903
C05022=1110.020,-81.390,-47.943,179.772,4.912,148.904
C05023=1110.015,-81.140,-47.954,179.772,4.917,148.905
C05024=1110.009,-80.890,-47.964,179.772,4.923,148.906
C05025=1110.004,-80.640,-47.975,179.772,4.928,148.907
C05026=1109.999,-80.391,-47.986,179.772,4.933,148.909
C05027=1109.994,-80.141,-47.996,179.771,4.938,148.910
C05028=1109.988,-79.892,-48.007,179.771,4.943,148.911
C05029=1109.983,-79.641,-48.018,179.771,4.948,148.912
C05030=1109.977,-79.392,-48.029,179.771,4.953,148.913
C05031=1109.972,-79.142,-48.040,179.771,4.959,148.915
C05032=1109.967,-78.892,-48.050,179.771,4.964,148.916
C05033=1109.962,-78.642,-48.061,179.770,4.969,148.917
C05034=1109.957,-78.393,-48.072,179.770,4.974,148.918
C05035=1109.952,-78.143,-48.082,179.770,4.979,148.919
C05036=1109.946,-77.894,-48.093,179.770,4.984,148.920
C05037=1109.941,-77.644,-48.104,179.770,4.989,148.922
C05038=1109.935,-77.394,-48.114,179.770,4.995,148.923
C05039=1109.930,-77.144,-48.126,179.770,5.000,148.924
C05040=1109.925,-76.895,-48.136,179.769,5.005,148.925
C05041=1109.920,-76.645,-48.147,179.769,5.010,148.926
C05042=1109.915,-76.395,-48.158,179.769,5.015,148.927
C05043=1109.910,-76.146,-48.169,179.769,5.020,148.929
C05044=1109.904,-75.895,-48.180,179.769,5.025,148.930
C05045=1109.899,-75.647,-48.191,179.769,5.031,148.931
C05046=1109.894,-75.396,-48.201,179.768,5.036,148.932
C05047=1109.888,-75.147,-48.212,179.768,5.041,148.933
C05048=1109.883,-74.897,-48.223,179.768,5.046,148.934
C05049=1109.878,-74.647,-48.235,179.768,5.051,148.936
C05050=1109.872,-74.398,-48.245,179.768,5.056,148.937
C05051=1109.868,-74.148,-48.256,179.768,5.061,148.938
C05052=1109.862,-73.898,-48.266,179.768,5.067,148.939
C05053=1109.857,-73.649,-48.278,179.767,5.072,148.940
C05054=1109.853,-73.433,-48.287,179.768,5.076,148.941
C05055=1109.848,-73.219,-48.297,179.768,5.080,148.942
C05056=1109.843,-73.004,-48.307,179.768,5.085,148.943
C05057=1109.839,-72.790,-48.315,179.768,5.089,148.944
C05058=1109.835,-72.575,-48.325,179.768,5.094,148.945
C05059=1109.830,-72.361,-48.335,179.767,5.098,148.946
C05060=1109.825,-72.146,-48.345,179.768,5.103,148.947
C05061=1109.821,-71.931,-48.353,179.768,5.108,148.948
C05062=1109.815,-71.682,-48.365,179.768,5.113,148.949
C05063=1109.811,-71.432,-48.376,179.768,5.118,148.950
C05064=1109.806,-71.182,-48.387,179.768,5.123,148.952
C05065=1109.800,-70.932,-48.398,179.768,5.128,148.952
C05066=1109.795,-70.682,-48.409,179.768,5.133,148.954
C05067=1109.790,-70.433,-48.420,179.768,5.138,148.955
C05068=1109.784,-70.183,-48.432,179.768,5.143,148.956
C05069=1109.779,-69.934,-48.443,179.768,5.148,148.957
C05070=1109.774,-69.683,-48.454,179.768,5.153,148.958
C05071=1109.768,-69.434,-48.465,179.768,5.159,148.959
C05072=1109.763,-69.185,-48.476,179.768,5.164,148.960
C05073=1109.758,-68.934,-48.487,179.769,5.169,148.961
C05074=1109.752,-68.685,-48.498,179.768,5.174,148.962
C05075=1109.748,-68.436,-48.510,179.768,5.179,148.964
C05076=1109.743,-68.186,-48.521,179.769,5.184,148.965
C05077=1109.737,-67.936,-48.532,179.769,5.189,148.966
C05078=1109.732,-67.686,-48.543,179.768,5.194,148.967
C05079=1109.727,-67.436,-48.555,179.769,5.200,148.968
C05080=1109.722,-67.187,-48.566,179.769,5.205,148.969
C05081=1109.716,-66.937,-48.576,179.769,5.210,148.970
C05082=1109.711,-66.687,-48.588,179.770,5.215,148.971
C05083=1109.706,-66.438,-48.600,179.769,5.220,148.972
C05084=1109.701,-66.188,-48.612,179.769,5.225,148.973
C05085=1109.695,-65.939,-48.622,179.770,5.231,148.974
C05086=1109.691,-65.689,-48.634,179.770,5.236,148.975
C05087=1109.685,-65.439,-48.645,179.771,5.241,148.976
C05088=1109.680,-65.189,-48.656,179.770,5.246,148.978
C05089=1109.674,-64.940,-48.668,179.771,5.251,148.978
C05090=1109.670,-64.690,-48.679,179.771,5.256,148.980
C05091=1109.664,-64.440,-48.691,179.771,5.260,148.981
C05092=1109.659,-64.191,-48.702,179.772,5.266,148.982
C05093=1109.654,-63.941,-48.714,179.772,5.271,148.983
C05094=1109.649,-63.692,-48.725,179.772,5.276,148.984
C05095=1109.643,-63.442,-48.737,179.772,5.281,148.985
C05096=1109.638,-63.192,-48.747,179.773,5.286,148.986
C05097=1109.633,-62.942,-48.759,179.772,5.291,148.987
C05098=1109.628,-62.692,-48.771,179.773,5.296,148.988
C05099=1109.622,-62.443,-48.782,179.773,5.302,148.989
C05100=1109.618,-62.193,-48.793,179.774,5.306,148.990
C05101=1109.612,-61.943,-48.805,179.774,5.311,148.991
C05102=1109.607,-61.694,-48.817,179.774,5.316,148.992
C05103=1109.602,-61.444,-48.829,179.775,5.322,148.993
C05104=1109.597,-61.194,-48.840,179.775,5.327,148.994
C05105=1109.591,-60.945,-48.851,179.775,5.332,148.995
C05106=1109.587,-60.695,-48.863,179.776,5.336,148.996
C05107=1109.581,-60.445,-48.874,179.776,5.341,148.997
C05108=1109.576,-60.195,-48.886,179.776,5.346,148.998
C05109=1109.571,-59.946,-48.898,179.777,5.352,148.999
C05110=1109.567,-59.731,-48.908,179.777,5.355,149.000
C05111=1109.562,-59.517,-48.918,179.777,5.359,149.000
C05112=1109.558,-59.302,-48.928,179.777,5.363,149.001
C05113=1109.553,-59.088,-48.938,179.777,5.367,149.002
C05114=1109.549,-58.873,-48.948,179.776,5.371,149.003
C05115=1109.544,-58.659,-48.958,179.776,5.375,149.004
C05116=1109.540,-58.444,-48.968,179.777,5.380,149.005
C05117=1109.536,-58.229,-48.978,179.776,5.384,149.006
C05118=1109.530,-57.980,-48.990,179.776,5.388,149.007
C05119=1109.526,-57.730,-49.002,179.776,5.393,149.008
C05120=1109.520,-57.480,-49.013,179.776,5.398,149.009
C05121=1109.514,-57.231,-49.025,179.775,5.402,149.010
C05122=1109.509,-56.981,-49.036,179.776,5.407,149.011
C05123=1109.504,-56.732,-49.049,179.775,5.412,149.013
C05124=1109.499,-56.482,-49.061,179.775,5.416,149.013
C05125=1109.494,-56.232,-49.072,179.775,5.421,149.015
C05126=1109.489,-55.982,-49.084,179.775,5.426,149.016
C05127=1109.483,-55.732,-49.096,179.775,5.430,149.017
C05128=1109.479,-55.483,-49.108,179.775,5.436,149.018
C05129=1109.474,-55.233,-49.120,179.774,5.440,149.019
C05130=1109.468,-54.983,-49.132,179.775,5.445,149.020
C05131=1109.463,-54.734,-49.143,179.775,5.450,149.021
C05132=1109.458,-54.484,-49.155,179.774,5.454,149.022
C05133=1109.453,-54.235,-49.167,179.774,5.459,149.023
C05134=1109.448,-53.985,-49.179,179.774,5.463,149.024
C05135=1109.443,-53.735,-49.191,179.774,5.468,149.025
C05136=1109.437,-53.485,-49.202,179.774,5.473,149.026
C05137=1109.432,-53.236,-49.215,179.773,5.477,149.028
C05138=1109.427,-52.987,-49.226,179.774,5.482,149.028
C05139=1109.421,-52.737,-49.238,179.774,5.487,149.030
C05140=1109.416,-52.487,-49.250,179.773,5.492,149.031
C05141=1109.411,-52.238,-49.262,179.773,5.496,149.032
C05142=1109.406,-51.988,-49.274,179.773,5.501,149.033
C05143=1109.401,-51.738,-49.286,179.773,5.506,149.034
C05144=1109.396,-51.489,-49.298,179.773,5.511,149.035
C05145=1109.390,-51.239,-49.310,179.772,5.515,149.036
C05146=1109.386,-50.989,-49.321,179.772,5.520,149.037
C05147=1109.380,-50.740,-49.334,179.773,5.525,149.038
C05148=1109.375,-50.490,-49.346,179.772,5.529,149.039
C05149=1109.370,-50.240,-49.358,179.772,5.534,149.040
C05150=1109.364,-49.991,-49.370,179.772,5.539,149.041
C05151=1109.359,-49.741,-49.382,179.772,5.543,149.042
C05152=1109.355,-49.492,-49.394,179.772,5.548,149.044
C05153=1109.349,-49.242,-49.406,179.771,5.554,149.045
C05154=1109.344,-48.992,-49.418,179.771,5.557,149.046
C05155=1109.339,-48.743,-49.431,179.771,5.563,149.047
C05156=1109.333,-48.493,-49.442,179.771,5.567,149.048
C05157=1109.328,-48.243,-49.455,179.771,5.572,149.049
C05158=1109.323,-47.994,-49.466,179.771,5.577,149.050
C05159=1109.318,-47.744,-49.478,179.770,5.581,149.051
C05160=1109.313,-47.494,-49.491,179.771,5.586,149.052
C05161=1109.308,-47.244,-49.503,179.771,5.591,149.053
C05162=1109.303,-46.994,-49.516,179.770,5.595,149.054
C05163=1109.297,-46.745,-49.528,179.770,5.600,149.056
C05164=1109.292,-46.495,-49.540,179.770,5.604,149.056
C05165=1109.288,-46.246,-49.551,179.770,5.610,149.058
C05166=1109.283,-46.031,-49.563,179.769,5.613,149.059
C05167=1109.279,-45.816,-49.573,179.769,5.617,149.059
C05168=1109.274,-45.603,-49.583,179.769,5.621,149.060
C05169=1109.270,-45.388,-49.593,179.769,5.625,149.061
C05170=1109.265,-45.173,-49.604,179.769,5.630,149.062
C05171=1109.260,-44.958,-49.614,179.769,5.634,149.063
C05172=1109.256,-44.744,-49.625,179.769,5.638,149.064
C05173=1109.252,-44.530,-49.636,179.768,5.642,149.065
C05174=1109.247,-44.280,-49.648,179.769,5.647,149.066
C05175=1109.242,-44.031,-49.660,179.768,5.651,149.067
C05176=1109.236,-43.781,-49.672,179.768,5.656,149.068
C05177=1109.231,-43.531,-49.685,179.767,5.661,149.070
C05178=1109.226,-43.281,-49.697,179.768,5.665,149.070
C05179=1109.221,-43.032,-49.709,179.768,5.671,149.072
C05180=1109.216,-42.781,-49.722,179.767,5.675,149.073
C05181=1109.211,-42.532,-49.734,179.768,5.680,149.074
C05182=1109.206,-42.283,-49.747,179.769,5.685,149.075
C05183=1109.200,-42.033,-49.759,179.769,5.690,149.075
C05184=1109.195,-41.784,-49.771,179.770,5.696,149.076
C05185=1109.190,-41.534,-49.784,179.771,5.700,149.077
C05186=1109.185,-41.284,-49.796,179.770,5.705,149.078
C05187=1109.179,-41.035,-49.808,179.771,5.710,149.079
C05188=1109.175,-40.784,-49.821,179.772,5.716,149.080
C05189=1109.169,-40.535,-49.833,179.772,5.720,149.081
C05190=1109.164,-40.286,-49.846,179.773,5.725,149.082
C05191=1109.159,-40.036,-49.858,179.773,5.730,149.083
C05192=1109.154,-39.787,-49.870,179.774,5.735,149.084
C05193=1109.149,-39.537,-49.883,179.774,5.739,149.085
C05194=1109.144,-39.287,-49.896,179.775,5.744,149.086
C05195=1109.139,-39.037,-49.908,179.775,5.749,149.087
C05196=1109.133,-38.788,-49.921,179.775,5.754,149.088
C05197=1109.128,-38.538,-49.934,179.777,5.759,149.088
C05198=1109.123,-38.289,-49.946,179.777,5.763,149.089
C05199=1109.117,-38.039,-49.958,179.778,5.768,149.090
C05200=1109.113,-37.789,-49.971,179.778,5.772,149.091
C05201=1109.108,-37.540,-49.984,179.778,5.777,149.092
C05202=1109.102,-37.290,-49.996,179.779,5.782,149.093
C05203=1109.097,-37.041,-50.009,179.779,5.786,149.094
C05204=1109.092,-36.790,-50.021,179.780,5.791,149.095
C05205=1109.087,-36.541,-50.034,179.780,5.796,149.096
C05206=1109.081,-36.291,-50.047,179.781,5.800,149.096
C05207=1109.076,-36.042,-50.059,179.781,5.805,149.097
C05208=1109.071,-35.793,-50.072,179.782,5.810,149.098
C05209=1109.067,-35.543,-50.085,179.782,5.814,149.099
C05210=1109.061,-35.293,-50.097,179.782,5.818,149.100
C05211=1109.055,-35.043,-50.110,179.783,5.823,149.101
C05212=1109.050,-34.794,-50.123,179.783,5.828,149.102
C05213=1109.046,-34.544,-50.136,179.784,5.832,149.102
C05214=1109.041,-34.295,-50.148,179.784,5.836,149.103
C05215=1109.035,-34.045,-50.161,179.784,5.841,149.104
C05216=1109.031,-33.795,-50.174,179.785,5.846,149.105
C05217=1109.025,-33.546,-50.187,179.785,5.850,149.106
C05218=1109.020,-33.296,-50.200,179.785,5.854,149.107
C05219=1109.015,-33.047,-50.212,179.785,5.859,149.108
C05220=1109.010,-32.797,-50.225,179.786,5.864,149.109
C05221=1109.004,-32.547,-50.238,179.786,5.867,149.109
C05222=1109.000,-32.333,-50.249,179.786,5.871,149.110
C05223=1108.996,-32.119,-50.260,179.787,5.876,149.111
C05224=1108.992,-31.904,-50.271,179.787,5.879,149.112
C05225=1108.987,-31.690,-50.282,179.787,5.883,149.113
C05226=1108.983,-31.476,-50.293,179.788,5.887,149.113
C05227=1108.978,-31.261,-50.304,179.787,5.890,149.114
C05228=1108.974,-31.047,-50.315,179.788,5.894,149.115
C05229=1108.969,-30.832,-50.327,179.788,5.898,149.116
C05230=1108.965,-30.582,-50.339,179.788,5.903,149.117
C05231=1108.960,-30.333,-50.352,179.788,5.907,149.118
C05232=1108.954,-30.083,-50.365,179.788,5.911,149.118
C05233=1108.949,-29.833,-50.378,179.789,5.916,149.119
C05234=1108.944,-29.584,-50.391,179.789,5.920,149.120
C05235=1108.938,-29.334,-50.404,179.789,5.925,149.121
C05236=1108.934,-29.084,-50.417,179.789,5.929,149.122
C05237=1108.929,-28.835,-50.430,179.790,5.933,149.123
C05238=1108.923,-28.586,-50.442,179.789,5.937,149.124
C05239=1108.918,-28.335,-50.456,179.790,5.942,149.125
C05240=1108.913,-28.086,-50.468,179.789,5.946,149.126
C05241=1108.908,-27.837,-50.482,179.790,5.951,149.127
C05242=1108.903,-27.587,-50.495,179.790,5.955,149.128
C05243=1108.898,-27.338,-50.508,179.790,5.960,149.129
C05244=1108.893,-27.087,-50.521,179.789,5.964,149.130
C05245=1108.888,-26.838,-50.534,179.790,5.969,149.131
C05246=1108.882,-26.589,-50.547,179.790,5.973,149.132
C05247=1108.877,-26.338,-50.560,179.790,5.978,149.133
C05248=1108.872,-26.090,-50.573,179.790,5.982,149.134
C05249=1108.868,-25.840,-50.586,179.790,5.987,149.135
C05250=1108.862,-25.590,-50.600,179.790,5.991,149.136
C05251=1108.857,-25.341,-50.612,179.790,5.996,149.137
C05252=1108.852,-25.090,-50.626,179.790,6.000,149.137
C05253=1108.847,-24.842,-50.639,179.791,6.005,149.138
C05254=1108.842,-24.592,-50.652,179.791,6.010,149.140
C05255=1108.836,-24.342,-50.665,179.791,6.015,149.140
C05256=1108.831,-24.093,-50.678,179.792,6.020,149.141
C05257=1108.826,-23.843,-50.692,179.792,6.024,149.142
C05258=1108.821,-23.594,-50.705,179.793,6.029,149.143
C05259=1108.816,-23.343,-50.718,179.793,6.034,149.144
C05260=1108.811,-23.094,-50.731,179.794,6.039,149.145
C05261=1108.806,-22.844,-50.745,179.794,6.043,149.146
C05262=1108.801,-22.595,-50.758,179.795,6.048,149.147
C05263=1108.796,-22.345,-50.771,179.795,6.053,149.148
C05264=1108.791,-22.096,-50.785,179.795,6.057,149.149
C05265=1108.785,-21.847,-50.797,179.795,6.062,149.150
C05266=1108.780,-21.596,-50.811,179.796,6.067,149.151
C05267=1108.775,-21.348,-50.824,179.796,6.071,149.151
C05268=1108.770,-21.097,-50.838,179.797,6.076,149.152
C05269=1108.765,-20.848,-50.850,179.797,6.081,149.153
C05270=1108.760,-20.598,-50.865,179.798,6.085,149.154
C05271=1108.754,-20.349,-50.878,179.798,6.090,149.155
C05272=1108.750,-20.099,-50.891,179.798,6.095,149.156
C05273=1108.744,-19.850,-50.905,179.799,6.100,149.157
C05274=1108.740,-19.600,-50.918,179.799,6.104,149.158
C05275=1108.734,-19.351,-50.932,179.800,6.108,149.158
C05276=1108.730,-19.101,-50.945,179.800,6.113,149.159
C05277=1108.724,-18.851,-50.958,179.801,6.117,149.160
C05278=1108.720,-18.636,-50.970,179.801,6.121,149.161
C05279=1108.716,-18.422,-50.981,179.802,6.126,149.162
C05280=1108.711,-18.208,-50.993,179.802,6.130,149.163
C05281=1108.707,-17.994,-51.004,179.802,6.134,149.163
C05282=1108.702,-17.780,-51.016,179.803,6.137,149.164
C05283=1108.697,-17.565,-51.028,179.803,6.141,149.165
C05284=1108.694,-17.351,-51.039,179.804,6.146,149.166
C05285=1108.689,-17.136,-51.051,179.804,6.149,149.166
C05286=1108.684,-16.887,-51.065,179.805,6.154,149.167
C05287=1108.679,-16.637,-51.078,179.805,6.159,149.168
C05288=1108.674,-16.388,-51.091,179.805,6.163,149.169
C05289=1108.668,-16.138,-51.105,179.805,6.167,149.170
C05290=1108.664,-15.888,-51.119,179.806,6.172,149.171
C05291=1108.658,-15.639,-51.132,179.806,6.177,149.172
C05292=1108.653,-15.389,-51.146,179.807,6.181,149.172
C05293=1108.648,-15.140,-51.159,179.808,6.186,149.173
C05294=1108.643,-14.890,-51.173,179.808,6.191,149.174
C05295=1108.638,-14.640,-51.187,179.809,6.195,149.175
C05296=1108.633,-14.391,-51.200,179.809,6.200,149.176
C05297=1108.628,-14.141,-51.214,179.809,6.204,149.177
C05298=1108.622,-13.892,-51.227,179.810,6.208,149.178
C05299=1108.618,-13.642,-51.241,179.811,6.213,149.178
C05300=1108.613,-13.393,-51.255,179.811,6.218,149.179
C05301=1108.607,-13.143,-51.269,179.812,6.222,149.180
C05302=1108.603,-12.894,-51.282,179.812,6.227,149.181
C05303=1108.598,-12.645,-51.296,179.813,6.232,149.182
C05304=1108.592,-12.394,-51.310,179.814,6.236,149.183
C05305=1108.587,-12.144,-51.324,179.814,6.240,149.184
C05306=1108.583,-11.896,-51.337,179.814,6.245,149.184
C05307=1108.577,-11.645,-51.351,179.815,6.250,149.185
C05308=1108.572,-11.396,-51.365,179.816,6.254,149.186
C05309=1108.567,-11.147,-51.379,179.816,6.259,149.187
C05310=1108.562,-10.897,-51.392,179.817,6.263,149.188
C05311=1108.557,-10.647,-51.406,179.817,6.268,149.189
C05312=1108.552,-10.398,-51.420,179.818,6.273,149.190
C05313=1108.547,-10.148,-51.434,179.818,6.276,149.190
C05314=1108.542,-9.899,-51.449,179.819,6.281,149.191
C05315=1108.537,-9.649,-51.461,179.819,6.286,149.192
C05316=1108.532,-9.400,-51.476,179.820,6.291,149.193
C05317=1108.527,-9.150,-51.490,179.821,6.295,149.194
C05318=1108.521,-8.901,-51.504,179.821,6.300,149.195
C05319=1108.516,-8.651,-51.517,179.822,6.304,149.195
C05320=1108.512,-8.401,-51.531,179.822,6.309,149.196
C05321=1108.507,-8.151,-51.545,179.822,6.313,149.197
C05322=1108.501,-7.902,-51.559,179.823,6.317,149.198
C05323=1108.496,-7.653,-51.574,179.823,6.322,149.199
C05324=1108.491,-7.403,-51.588,179.824,6.327,149.200
C05325=1108.486,-7.154,-51.602,179.825,6.331,149.200
C05326=1108.481,-6.904,-51.615,179.825,6.336,149.201
C05327=1108.476,-6.654,-51.629,179.826,6.340,149.202
C05328=1108.471,-6.405,-51.643,179.827,6.345,149.203
C05329=1108.466,-6.156,-51.657,179.827,6.349,149.204
C05330=1108.461,-5.906,-51.671,179.827,6.353,149.205
C05331=1108.456,-5.656,-51.686,179.828,6.358,149.205
C05332=1108.451,-5.406,-51.700,179.829,6.362,149.206
C05333=1108.445,-5.157,-51.714,179.829,6.367,149.207
C05334=1108.442,-4.943,-51.726,179.830,6.371,149.208
C05335=1108.437,-4.729,-51.738,179.831,6.375,149.208
C05336=1108.433,-4.515,-51.750,179.831,6.379,149.209
C05337=1108.429,-4.300,-51.762,179.831,6.383,149.210
C05338=1108.424,-4.086,-51.774,179.832,6.387,149.211
C05339=1108.420,-3.872,-51.786,179.832,6.390,149.211
C05340=1108.416,-3.657,-51.798,179.833,6.394,149.212
C05341=1108.411,-3.443,-51.811,179.833,6.399,149.213
C05342=1108.406,-3.193,-51.825,179.834,6.403,149.214
C05343=1108.401,-2.944,-51.839,179.834,6.407,149.214
C05344=1108.396,-2.695,-51.853,179.835,6.412,149.215
C05345=1108.391,-2.445,-51.867,179.836,6.416,149.216
C05346=1108.386,-2.195,-51.882,179.836,6.421,149.217
C05347=1108.381,-1.946,-51.896,179.837,6.425,149.218
C05348=1108.376,-1.696,-51.910,179.837,6.430,149.219
C05349=1108.371,-1.447,-51.926,179.838,6.434,149.219
C05350=1108.365,-1.198,-51.940,179.839,6.439,149.220
C05351=1108.360,-0.948,-51.954,179.839,6.444,149.221
C05352=1108.355,-0.698,-51.968,179.840,6.448,149.222
C05353=1108.350,-0.448,-51.982,179.841,6.453,149.223
C05354=1108.345,-0.199,-51.997,179.841,6.457,149.224
C05355=1108.340,0.051,-52.011,179.842,6.461,149.224
C05356=1108.335,0.300,-52.025,179.842,6.466,149.225
C05357=1108.330,0.549,-52.040,179.843,6.471,149.226
C05358=1108.325,0.799,-52.054,179.843,6.475,149.227
C05359=1108.320,1.049,-52.068,179.844,6.480,149.228
C05360=1108.315,1.298,-52.083,179.845,6.484,149.228
C05361=1108.310,1.548,-52.097,179.846,6.489,149.229
C05362=1108.305,1.798,-52.111,179.846,6.494,149.230
C05363=1108.301,2.047,-52.126,179.847,6.498,149.231
C05364=1108.294,2.296,-52.141,179.848,6.503,149.232
C05365=1108.289,2.546,-52.155,179.848,6.508,149.233
C05366=1108.284,2.796,-52.169,179.849,6.512,149.233
C05367=1108.280,3.045,-52.184,179.850,6.517,149.234
C05368=1108.275,3.294,-52.199,179.850,6.520,149.235
C05369=1108.270,3.544,-52.213,179.850,6.525,149.236
C05370=1108.265,3.794,-52.227,179.851,6.530,149.237
C05371=1108.260,4.043,-52.243,179.852,6.534,149.238
C05372=1108.255,4.293,-52.257,179.852,6.539,149.238
C05373=1108.250,4.543,-52.271,179.853,6.544,149.239
C05374=1108.245,4.792,-52.286,179.854,6.548,149.240
C05375=1108.240,5.041,-52.301,179.854,6.553,149.241
C05376=1108.234,5.291,-52.315,179.855,6.557,149.242
C05377=1108.229,5.540,-52.330,179.855,6.562,149.243
C05378=1108.224,5.789,-52.344,179.856,6.566,149.243
C05379=1108.219,6.039,-52.359,179.857,6.571,149.244
C05380=1108.215,6.288,-52.374,179.858,6.576,149.245
C05381=1108.209,6.538,-52.388,179.858,6.581,149.246
C05382=1108.204,6.787,-52.403,179.859,6.585,149.247
C05383=1108.199,7.037,-52.418,179.860,6.590,149.248
C05384=1108.194,7.287,-52.432,179.860,6.594,149.248
C05385=1108.189,7.536,-52.448,179.861,6.599,149.249
C05386=1108.184,7.786,-52.462,179.861,6.604,149.250
C05387=1108.179,8.035,-52.477,179.862,6.608,149.251
C05388=1108.174,8.285,-52.491,179.863,6.613,149.252
C05389=1108.169,8.534,-52.507,179.863,6.617,149.253
C05390=1108.165,8.749,-52.519,179.863,6.621,149.254
C05391=1108.161,8.963,-52.531,179.864,6.625,149.254
C05392=1108.156,9.177,-52.545,179.865,6.629,149.255
C05393=1108.152,9.391,-52.557,179.865,6.633,149.256
C05394=1108.148,9.605,-52.571,179.865,6.637,149.256
C05395=1108.143,9.819,-52.583,179.865,6.640,149.257
C05396=1108.139,10.034,-52.595,179.866,6.645,149.258
C05397=1108.134,10.247,-52.608,179.866,6.648,149.259
C05398=1108.129,10.497,-52.623,179.867,6.653,149.259
C05399=1108.125,10.746,-52.638,179.867,6.657,149.260
C05400=1108.119,10.996,-52.653,179.867,6.662,149.261
C05401=1108.114,11.245,-52.668,179.868,6.666,149.262
C05402=1108.110,11.495,-52.683,179.869,6.671,149.263
C05403=1108.105,11.745,-52.698,179.869,6.675,149.264
C05404=1108.100,11.994,-52.713,179.870,6.679,149.265
C05405=1108.094,12.244,-52.728,179.870,6.684,149.265
C05406=1108.090,12.493,-52.743,179.871,6.689,149.266
C05407=1108.085,12.742,-52.758,179.871,6.694,149.267
C05408=1108.079,12.993,-52.772,179.872,6.697,149.268
C05409=1108.075,13.242,-52.787,179.872,6.702,149.269
C05410=1108.069,13.491,-52.803,179.873,6.706,149.270
C05411=1108.064,13.741,-52.817,179.873,6.711,149.271
C05412=1108.060,13.990,-52.832,179.873,6.715,149.271
C05413=1108.054,14.239,-52.848,179.874,6.719,149.272
C05414=1108.049,14.489,-52.862,179.875,6.724,149.273
C05415=1108.045,14.739,-52.878,179.875,6.729,149.274
C05416=1108.040,14.988,-52.893,179.876,6.732,149.275
C05417=1108.034,15.238,-52.908,179.876,6.737,149.275
C05418=1108.030,15.487,-52.923,179.877,6.742,149.276
C05419=1108.024,15.737,-52.939,179.877,6.746,149.277
C05420=1108.020,15.986,-52.954,179.878,6.750,149.278
C05421=1108.014,16.236,-52.968,179.878,6.755,149.279
C05422=1108.009,16.485,-52.983,179.879,6.759,149.280
C05423=1108.004,16.735,-52.999,179.880,6.764,149.280
C05424=1108.000,16.984,-53.014,179.880,6.768,149.281
C05425=1107.994,17.234,-53.029,179.881,6.772,149.282
C05426=1107.989,17.483,-53.044,179.882,6.777,149.283
C05427=1107.984,17.733,-53.060,179.882,6.781,149.284
C05428=1107.979,17.982,-53.075,179.883,6.785,149.284
C05429=1107.975,18.232,-53.091,179.883,6.790,149.285
C05430=1107.970,18.481,-53.105,179.884,6.794,149.286
C05431=1107.964,18.731,-53.121,179.885,6.799,149.287
C05432=1107.960,18.980,-53.136,179.885,6.802,149.288
C05433=1107.954,19.229,-53.151,179.886,6.807,149.288
C05434=1107.950,19.478,-53.166,179.886,6.811,149.289
C05435=1107.945,19.729,-53.182,179.887,6.816,149.290
C05436=1107.939,19.978,-53.198,179.887,6.820,149.291
C05437=1107.935,20.227,-53.213,179.888,6.824,149.292
C05438=1107.929,20.477,-53.228,179.889,6.829,149.292
C05439=1107.924,20.726,-53.243,179.890,6.833,149.293
C05440=1107.920,20.976,-53.259,179.890,6.837,149.294
C05441=1107.914,21.226,-53.274,179.891,6.842,149.295
C05442=1107.910,21.475,-53.289,179.892,6.846,149.295
C05443=1107.904,21.724,-53.305,179.892,6.851,149.296
C05444=1107.900,21.974,-53.320,179.893,6.854,149.297
C05445=1107.895,22.223,-53.336,179.894,6.859,149.297
C05446=1107.890,22.437,-53.349,179.894,6.862,149.298
C05447=1107.886,22.651,-53.362,179.895,6.866,149.299
C05448=1107.882,22.865,-53.376,179.896,6.870,149.299
C05449=1107.877,23.080,-53.388,179.896,6.873,149.300
C05450=1107.873,23.294,-53.402,179.896,6.877,149.301
C05451=1107.869,23.508,-53.415,179.897,6.880,149.301
C05452=1107.865,23.722,-53.429,179.898,6.885,149.302
C05453=1107.861,23.935,-53.442,179.898,6.888,149.303
C05454=1107.855,24.185,-53.457,179.899,6.893,149.303
C05455=1107.850,24.435,-53.473,179.899,6.896,149.304
C05456=1107.846,24.684,-53.488,179.900,6.901,149.305
C05457=1107.840,24.933,-53.504,179.901,6.906,149.306
C05458=1107.836,25.184,-53.520,179.901,6.909,149.306
C05459=1107.830,25.433,-53.535,179.902,6.913,149.307
C05460=1107.825,25.682,-53.550,179.903,6.918,149.308
C05461=1107.820,25.931,-53.566,179.904,6.922,149.309
C05462=1107.816,26.181,-53.583,179.904,6.926,149.309
C05463=1107.811,26.430,-53.598,179.905,6.931,149.310
C05464=1107.806,26.679,-53.613,179.906,6.935,149.311
C05465=1107.801,26.930,-53.629,179.907,6.939,149.312
C05466=1107.795,27.179,-53.645,179.907,6.943,149.312
C05467=1107.790,27.428,-53.660,179.908,6.947,149.313
C05468=1107.786,27.678,-53.676,179.909,6.952,149.314
C05469=1107.781,27.927,-53.692,179.910,6.956,149.314
C05470=1107.776,28.176,-53.708,179.910,6.960,149.315
C05471=1107.771,28.426,-53.724,179.911,6.964,149.316
C05472=1107.765,28.676,-53.739,179.912,6.969,149.317
C05473=1107.761,28.925,-53.754,179.913,6.972,149.317
C05474=1107.756,29.174,-53.771,179.913,6.977,149.318
C05475=1107.751,29.424,-53.786,179.914,6.981,149.319
C05476=1107.745,29.673,-53.802,179.916,6.985,149.319
C05477=1107.741,29.923,-53.818,179.916,6.989,149.320
C05478=1107.736,30.172,-53.834,179.917,6.994,149.321
C05479=1107.732,30.422,-53.850,179.918,6.998,149.322
C05480=1107.726,30.671,-53.865,179.919,7.002,149.322
C05481=1107.721,30.920,-53.882,179.919,7.006,149.323
C05482=1107.716,31.170,-53.897,179.920,7.010,149.324
C05483=1107.711,31.420,-53.913,179.921,7.014,149.324
C05484=1107.706,31.670,-53.929,179.922,7.019,149.325
C05485=1107.701,31.919,-53.945,179.922,7.023,149.326
C05486=1107.696,32.168,-53.960,179.923,7.027,149.326
C05487=1107.692,32.418,-53.976,179.924,7.031,149.327
C05488=1107.686,32.666,-53.993,179.925,7.035,149.328
C05489=1107.682,32.917,-54.009,179.926,7.039,149.328
C05490=1107.677,33.165,-54.025,179.927,7.043,149.329
C05491=1107.671,33.415,-54.040,179.928,7.048,149.330
C05492=1107.666,33.665,-54.056,179.928,7.052,149.331
C05493=1107.661,33.914,-54.073,179.929,7.056,149.331
C05494=1107.657,34.164,-54.089,179.930,7.060,149.332
C05495=1107.652,34.413,-54.105,179.931,7.064,149.333
C05496=1107.647,34.663,-54.121,179.932,7.068,149.333
C05497=1107.642,34.911,-54.137,179.933,7.072,149.334
C05498=1107.637,35.162,-54.153,179.934,7.077,149.335
C05499=1107.631,35.411,-54.169,179.935,7.081,149.335
C05500=1107.626,35.660,-54.185,179.935,7.084,149.336
C05501=1107.622,35.910,-54.201,179.936,7.089,149.336
C05502=1107.618,36.124,-54.215,179.937,7.092,149.337
C05503=1107.613,36.338,-54.229,179.938,7.095,149.338
C05504=1107.608,36.551,-54.242,179.939,7.100,149.338
C05505=1107.604,36.765,-54.257,179.939,7.103,149.339
C05506=1107.601,36.979,-54.270,179.940,7.106,149.339
C05507=1107.597,37.194,-54.284,179.941,7.110,149.340
C05508=1107.593,37.407,-54.298,179.942,7.114,149.340
C05509=1107.588,37.622,-54.312,179.943,7.117,149.341
C05510=1107.583,37.870,-54.328,179.943,7.121,149.342
C05511=1107.578,38.120,-54.344,179.944,7.125,149.342
C05512=1107.573,38.370,-54.361,179.945,7.129,149.343
C05513=1107.568,38.620,-54.377,179.946,7.134,149.344
C05514=1107.563,38.868,-54.393,179.947,7.137,149.344
C05515=1107.558,39.118,-54.410,179.948,7.142,149.345
C05516=1107.553,39.367,-54.426,179.949,7.146,149.346
C05517=1107.548,39.617,-54.442,179.950,7.150,149.346
C05518=1107.543,39.866,-54.458,179.950,7.154,149.347
C05519=1107.539,40.116,-54.474,179.952,7.158,149.347
C05520=1107.533,40.364,-54.491,179.953,7.162,149.348
C05521=1107.529,40.615,-54.507,179.954,7.166,149.349
C05522=1107.523,40.864,-54.524,179.954,7.170,149.349
C05523=1107.518,41.113,-54.540,179.956,7.174,149.350
C05524=1107.514,41.363,-54.556,179.957,7.178,149.351
C05525=1107.509,41.612,-54.573,179.958,7.183,149.351
C05526=1107.504,41.861,-54.589,179.958,7.186,149.352
C05527=1107.499,42.110,-54.605,179.959,7.190,149.353
C05528=1107.493,42.361,-54.622,179.961,7.194,149.353
C05529=1107.489,42.610,-54.639,179.962,7.199,149.354
C05530=1107.484,42.859,-54.655,179.962,7.202,149.354
C05531=1107.479,43.108,-54.672,179.963,7.206,149.355
C05532=1107.474,43.358,-54.687,179.964,7.211,149.356
